LIN {X 0,Y 530.252,Z 278.433,A -85,B 0,C 180,E1 -4543.36,E2 -4543.36} C_VEL
LIN {X 0,Y 527.412,Z 278.789,A -85,B 0,C 180,E1 -4544.388,E2 -4544.388} C_VEL
LIN {X 0,Y 525.021,Z 279.084,A -85,B 0,C 180,E1 -4545.217,E2 -4545.217} C_VEL
LIN {X 0,Y 523.993,Z 279.212,A -85,B 0,C 180,E1 -4545.856,E2 -4545.856} C_VEL
LIN {X 0,Y 523.909,Z 279.223,A -85,B 0,C 180,E1 -4546.072,E2 -4546.072} C_VEL
LIN {X 0,Y 523.934,Z 279.22,A -85,B 0,C 180,E1 -4548.907,E2 -4548.907} C_VEL
LIN {X 0,Y 523.909,Z 279.226,A -85,B 0,C 180,E1 -4551.897,E2 -4551.897} C_VEL
LIN {X 0,Y 523.93,Z 279.219,A -85,B 0,C 180,E1 -4554.908,E2 -4554.908} C_VEL
LIN {X 0,Y 523.934,Z 279.224,A -85,B 0,C 180,E1 -4557.677,E2 -4557.677} C_VEL
LIN {X 0,Y 523.96,Z 279.215,A -85,B 0,C 180,E1 -4560.672,E2 -4560.672} C_VEL
LIN {X 0,Y 523.968,Z 279.22,A -85,B 0,C 180,E1 -4563.728,E2 -4563.728} C_VEL
LIN {X 0,Y 523.926,Z 279.22,A -85,B 0,C 180,E1 -4566.27,E2 -4566.27} C_VEL
LIN {X 0,Y 523.937,Z 279.221,A -85,B 0,C 180,E1 -4568.766,E2 -4568.766} C_VEL
LIN {X 0,Y 523.943,Z 279.222,A -85,B 0,C 180,E1 -4571.22,E2 -4571.22} C_VEL
LIN {X 0,Y 523.925,Z 279.22,A -85,B 0,C 180,E1 -4573.638,E2 -4573.638} C_VEL
LIN {X 0,Y 523.928,Z 279.219,A -85,B 0,C 180,E1 -4576.028,E2 -4576.028} C_VEL
LIN {X 0,Y 524,Z 279.215,A -85,B 0,C 180,E1 -4578.394,E2 -4578.394} C_VEL
LIN {X 0,Y 523.986,Z 279.211,A -85,B 0,C 180,E1 -4581.516,E2 -4581.516} C_VEL
LIN {X 0,Y 524.058,Z 279.206,A -85,B 0,C 180,E1 -4584.613,E2 -4584.613} C_VEL
LIN {X 0,Y 524.093,Z 279.2,A -85,B 0,C 180,E1 -4587.694,E2 -4587.694} C_VEL
LIN {X 0,Y 524.084,Z 279.207,A -85,B 0,C 180,E1 -4590,E2 -4590} C_VEL
LIN {X 0,Y 524.093,Z 279.2,A -85,B 0,C 180,E1 -4592.306,E2 -4592.306} C_VEL
LIN {X 0,Y 524.059,Z 279.206,A -85,B 0,C 180,E1 -4595.387,E2 -4595.387} C_VEL
LIN {X 0,Y 523.986,Z 279.211,A -85,B 0,C 180,E1 -4598.484,E2 -4598.484} C_VEL
LIN {X 0,Y 523.99,Z 279.214,A -85,B 0,C 180,E1 -4601.74,E2 -4601.74} C_VEL
LIN {X 0,Y 523.981,Z 279.218,A -85,B 0,C 180,E1 -4605.053,E2 -4605.053} C_VEL
LIN {X 0,Y 523.953,Z 279.216,A -85,B 0,C 180,E1 -4607.969,E2 -4607.969} C_VEL
LIN {X 0,Y 523.962,Z 279.218,A -85,B 0,C 180,E1 -4610.411,E2 -4610.411} C_VEL
LIN {X 0,Y 523.906,Z 279.227,A -85,B 0,C 180,E1 -4612.894,E2 -4612.894} C_VEL
LIN {X 0,Y 523.945,Z 279.217,A -85,B 0,C 180,E1 -4615.419,E2 -4615.419} C_VEL
LIN {X 0,Y 523.961,Z 279.219,A -85,B 0,C 180,E1 -4618,E2 -4618} C_VEL
LIN {X 0,Y 523.943,Z 279.219,A -85,B 0,C 180,E1 -4620.857,E2 -4620.857} C_VEL
LIN {X 0,Y 523.954,Z 279.22,A -85,B 0,C 180,E1 -4623.736,E2 -4623.736} C_VEL
LIN {X 0,Y 523.914,Z 279.223,A -85,B 0,C 180,E1 -4626.405,E2 -4626.405} C_VEL
LIN {X 0,Y 523.915,Z 279.222,A -85,B 0,C 180,E1 -4629.086,E2 -4629.086} C_VEL
LIN {X 0,Y 523.945,Z 279.219,A -85,B 0,C 180,E1 -4632.12,E2 -4632.12} C_VEL
LIN {X 0,Y 523.931,Z 279.226,A -85,B 0,C 180,E1 -4635.312,E2 -4635.312} C_VEL
LIN {X 0,Y 523.932,Z 279.22,A -85,B 0,C 180,E1 -4638.693,E2 -4638.693} C_VEL
LIN {X 0,Y 523.906,Z 279.221,A -85,B 0,C 180,E1 -4641.899,E2 -4641.899} C_VEL
LIN {X 0,Y 523.908,Z 279.227,A -85,B 0,C 180,E1 -4644.914,E2 -4644.914} C_VEL
LIN {X 0,Y 523.925,Z 279.218,A -85,B 0,C 180,E1 -4647.682,E2 -4647.682} C_VEL
LIN {X 0,Y 524.01,Z 279.336,A -85,B 0,C 180,E1 -4650.028,E2 -4650.028} C_VEL
LIN {X 0,Y 523.881,Z 285.472,A -85,B 0,C 180,E1 -4652.865,E2 -4652.865} C_VEL
LIN {X 0,Y 523.769,Z 291.976,A -85,B 0,C 180,E1 -4655.844,E2 -4655.844} C_VEL
LIN {X 0,Y 523.697,Z 298.443,A -85,B 0,C 180,E1 -4658.757,E2 -4658.757} C_VEL
LIN {X 0,Y 523.615,Z 303.894,A -85,B 0,C 180,E1 -4661.209,E2 -4661.209} C_VEL
LIN {X 0,Y 523.527,Z 309.386,A -85,B 0,C 180,E1 -4663.627,E2 -4663.627} C_VEL
LIN {X 0,Y 523.496,Z 314.819,A -85,B 0,C 180,E1 -4666.017,E2 -4666.017} C_VEL
LIN {X 0,Y 523.482,Z 320.596,A -85,B 0,C 180,E1 -4668.54,E2 -4668.54} C_VEL
LIN {X 0,Y 523.415,Z 328.516,A -85,B 0,C 180,E1 -4671.969,E2 -4671.969} C_VEL
LIN {X 0,Y 524.16,Z 336.561,A -85,B 0,C 180,E1 -4672.296,E2 -4672.296} C_VEL
LIN {X 0,Y 523.983,Z 346.121,A -85,B 0,C 180,E1 -4672.807,E2 -4672.807} C_VEL
LIN {X 0,Y 523.913,Z 353.385,A -85,B 0,C 180,E1 -4673.324,E2 -4673.324} C_VEL
LIN {X 0,Y 523.776,Z 359.239,A -85,B 0,C 180,E1 -4673.839,E2 -4673.839} C_VEL
LIN {X 0,Y 523.715,Z 366.141,A -85,B 0,C 180,E1 -4674.611,E2 -4674.611} C_VEL
LIN {X 0,Y 523.612,Z 371.545,A -85,B 0,C 180,E1 -4675.382,E2 -4675.382} C_VEL
LIN {X 0,Y 523.571,Z 375.823,A -85,B 0,C 180,E1 -4676.153,E2 -4676.153} C_VEL
LIN {X 0,Y 523.482,Z 379.147,A -85,B 0,C 180,E1 -4676.923,E2 -4676.923} C_VEL
LIN {X 0,Y 523.384,Z 381.639,A -85,B 0,C 180,E1 -4677.692,E2 -4677.692} C_VEL
LIN {X 0,Y 523.335,Z 383.365,A -85,B 0,C 180,E1 -4678.462,E2 -4678.462} C_VEL
LIN {X 0,Y 523.326,Z 384.379,A -85,B 0,C 180,E1 -4679.232,E2 -4679.232} C_VEL
LIN {X 0,Y 523.327,Z 384.776,A -85,B 0,C 180,E1 -4680.001,E2 -4680.001} C_VEL
LIN {X 0,Y 523.33,Z 384.536,A -85,B 0,C 180,E1 -4680.77,E2 -4680.77} C_VEL
LIN {X 0,Y 523.344,Z 383.632,A -85,B 0,C 180,E1 -4681.54,E2 -4681.54} C_VEL
LIN {X 0,Y 523.49,Z 380.907,A -85,B 0,C 180,E1 -4682.694,E2 -4682.694} C_VEL
LIN {X 0,Y 523.588,Z 378.19,A -85,B 0,C 180,E1 -4683.464,E2 -4683.464} C_VEL
LIN {X 0,Y 523.626,Z 373.539,A -85,B 0,C 180,E1 -4684.427,E2 -4684.427} C_VEL
LIN {X 0,Y 523.724,Z 368.666,A -85,B 0,C 180,E1 -4685.198,E2 -4685.198} C_VEL
LIN {X 0,Y 523.808,Z 362.441,A -85,B 0,C 180,E1 -4685.969,E2 -4685.969} C_VEL
LIN {X 0,Y 523.994,Z 354.754,A -85,B 0,C 180,E1 -4686.702,E2 -4686.702} C_VEL
LIN {X 0,Y 524.043,Z 346.949,A -85,B 0,C 180,E1 -4687.282,E2 -4687.282} C_VEL
LIN {X 0,Y 524.218,Z 337.48,A -85,B 0,C 180,E1 -4687.802,E2 -4687.802} C_VEL
LIN {X 0,Y 523.898,Z 331.555,A -85,B 0,C 180,E1 -4688.05,E2 -4688.05} C_VEL
LIN {X 0,Y 523.497,Z 329.053,A -85,B 0,C 180,E1 -4688.153,E2 -4688.153} C_VEL
LIN {X 0,Y 523.539,Z 321.18,A -85,B 0,C 180,E1 -4691.617,E2 -4691.617} C_VEL
LIN {X 0,Y 523.658,Z 313.899,A -85,B 0,C 180,E1 -4694.914,E2 -4694.914} C_VEL
LIN {X 0,Y 523.734,Z 307.092,A -85,B 0,C 180,E1 -4697.978,E2 -4697.978} C_VEL
LIN {X 0,Y 523.84,Z 301.836,A -85,B 0,C 180,E1 -4700.416,E2 -4700.416} C_VEL
LIN {X 0,Y 523.889,Z 296.392,A -85,B 0,C 180,E1 -4702.895,E2 -4702.895} C_VEL
LIN {X 0,Y 524.057,Z 289.588,A -85,B 0,C 180,E1 -4706.035,E2 -4706.035} C_VEL
LIN {X 0,Y 524.173,Z 283.477,A -85,B 0,C 180,E1 -4708.861,E2 -4708.861} C_VEL
LIN {X 0,Y 523.971,Z 279.222,A -85,B 0,C 180,E1 -4710.918,E2 -4710.918} C_VEL
LIN {X 0,Y 523.965,Z 279.222,A -85,B 0,C 180,E1 -4713.735,E2 -4713.735} C_VEL
LIN {X 0,Y 523.909,Z 279.227,A -85,B 0,C 180,E1 -4716.402,E2 -4716.402} C_VEL
LIN {X 0,Y 523.925,Z 279.227,A -85,B 0,C 180,E1 -4719.085,E2 -4719.085} C_VEL
LIN {X 0,Y 523.957,Z 279.222,A -85,B 0,C 180,E1 -4722.119,E2 -4722.119} C_VEL
LIN {X 0,Y 523.949,Z 279.223,A -85,B 0,C 180,E1 -4725.31,E2 -4725.31} C_VEL
LIN {X 0,Y 523.961,Z 279.222,A -85,B 0,C 180,E1 -4728.69,E2 -4728.69} C_VEL
LIN {X 0,Y 523.921,Z 279.226,A -85,B 0,C 180,E1 -4731.081,E2 -4731.081} C_VEL
LIN {X 0,Y 523.905,Z 279.229,A -85,B 0,C 180,E1 -4733.825,E2 -4733.825} C_VEL
LIN {X 0,Y 523.946,Z 279.225,A -85,B 0,C 180,E1 -4736.636,E2 -4736.636} C_VEL
LIN {X 0,Y 523.932,Z 279.256,A -85,B 0,C 180,E1 -4738.791,E2 -4738.791} C_VEL
LIN {X 0,Y 525.748,Z 287.197,A -85,B 0,C 180,E1 -4740.835,E2 -4740.835} C_VEL
LIN {X 0,Y 526.442,Z 291.224,A -85,B 0,C 180,E1 -4741.776,E2 -4741.776} C_VEL
LIN {X 0,Y 525.737,Z 304.415,A -85,B 0,C 180,E1 -4744.462,E2 -4744.462} C_VEL
LIN {X 0,Y 525.131,Z 318.686,A -85,B 0,C 180,E1 -4747.163,E2 -4747.163} C_VEL
LIN {X 0,Y 524.702,Z 334.54,A -85,B 0,C 180,E1 -4750.028,E2 -4750.028} C_VEL
LIN {X 0,Y 524.357,Z 350.704,A -85,B 0,C 180,E1 -4752.85,E2 -4752.85} C_VEL
LIN {X 0,Y 524.062,Z 369.627,A -85,B 0,C 180,E1 -4756.031,E2 -4756.031} C_VEL
LIN {X 0,Y 524.024,Z 371.591,A -85,B 0,C 180,E1 -4756.339,E2 -4756.339} C_VEL
LIN {X 0,Y 525.306,Z 382.111,A -85,B 0,C 180,E1 -4756.558,E2 -4756.558} C_VEL
LIN {X 0,Y 525.125,Z 394.093,A -85,B 0,C 180,E1 -4756.898,E2 -4756.898} C_VEL
LIN {X 0,Y 524.847,Z 407.07,A -85,B 0,C 180,E1 -4757.432,E2 -4757.432} C_VEL
LIN {X 0,Y 524.626,Z 419.038,A -85,B 0,C 180,E1 -4758.09,E2 -4758.09} C_VEL
LIN {X 0,Y 524.366,Z 430.416,A -85,B 0,C 180,E1 -4758.892,E2 -4758.892} C_VEL
LIN {X 0,Y 524.109,Z 440.369,A -85,B 0,C 180,E1 -4759.766,E2 -4759.766} C_VEL
LIN {X 0,Y 523.897,Z 449.423,A -85,B 0,C 180,E1 -4760.736,E2 -4760.736} C_VEL
LIN {X 0,Y 523.699,Z 458.25,A -85,B 0,C 180,E1 -4761.899,E2 -4761.899} C_VEL
LIN {X 0,Y 523.576,Z 465.285,A -85,B 0,C 180,E1 -4763.061,E2 -4763.061} C_VEL
LIN {X 0,Y 523.524,Z 470.919,A -85,B 0,C 180,E1 -4764.221,E2 -4764.221} C_VEL
LIN {X 0,Y 523.361,Z 475.325,A -85,B 0,C 180,E1 -4765.379,E2 -4765.379} C_VEL
LIN {X 0,Y 523.444,Z 477.673,A -85,B 0,C 180,E1 -4766.151,E2 -4766.151} C_VEL
LIN {X 0,Y 523.368,Z 479.561,A -85,B 0,C 180,E1 -4766.921,E2 -4766.921} C_VEL
LIN {X 0,Y 523.336,Z 480.978,A -85,B 0,C 180,E1 -4767.691,E2 -4767.691} C_VEL
LIN {X 0,Y 523.25,Z 482.598,A -85,B 0,C 180,E1 -4769.23,E2 -4769.23} C_VEL
LIN {X 0,Y 523.246,Z 482.818,A -85,B 0,C 180,E1 -4770,E2 -4770} C_VEL
LIN {X 0,Y 523.25,Z 482.599,A -85,B 0,C 180,E1 -4770.77,E2 -4770.77} C_VEL
LIN {X 0,Y 523.336,Z 480.979,A -85,B 0,C 180,E1 -4772.309,E2 -4772.309} C_VEL
LIN {X 0,Y 523.368,Z 479.563,A -85,B 0,C 180,E1 -4773.079,E2 -4773.079} C_VEL
LIN {X 0,Y 523.425,Z 476.591,A -85,B 0,C 180,E1 -4774.235,E2 -4774.235} C_VEL
LIN {X 0,Y 523.464,Z 472.56,A -85,B 0,C 180,E1 -4775.393,E2 -4775.393} C_VEL
LIN {X 0,Y 523.524,Z 467.22,A -85,B 0,C 180,E1 -4776.58,E2 -4776.58} C_VEL
LIN {X 0,Y 523.666,Z 460.813,A -85,B 0,C 180,E1 -4777.713,E2 -4777.713} C_VEL
LIN {X 0,Y 523.846,Z 452.653,A -85,B 0,C 180,E1 -4778.875,E2 -4778.875} C_VEL
LIN {X 0,Y 524.015,Z 444.319,A -85,B 0,C 180,E1 -4779.846,E2 -4779.846} C_VEL
LIN {X 0,Y 524.305,Z 434.143,A -85,B 0,C 180,E1 -4780.816,E2 -4780.816} C_VEL
LIN {X 0,Y 524.583,Z 422.543,A -85,B 0,C 180,E1 -4781.694,E2 -4781.694} C_VEL
LIN {X 0,Y 524.803,Z 411.237,A -85,B 0,C 180,E1 -4782.373,E2 -4782.373} C_VEL
LIN {X 0,Y 524.996,Z 399.713,A -85,B 0,C 180,E1 -4782.908,E2 -4782.908} C_VEL
LIN {X 0,Y 525.219,Z 386.487,A -85,B 0,C 180,E1 -4783.346,E2 -4783.346} C_VEL
LIN {X 0,Y 525.058,Z 379.612,A -85,B 0,C 180,E1 -4783.513,E2 -4783.513} C_VEL
LIN {X 0,Y 524.023,Z 371.416,A -85,B 0,C 180,E1 -4783.698,E2 -4783.698} C_VEL
LIN {X 0,Y 524.364,Z 353.595,A -85,B 0,C 180,E1 -4786.748,E2 -4786.748} C_VEL
LIN {X 0,Y 524.721,Z 336.251,A -85,B 0,C 180,E1 -4789.767,E2 -4789.767} C_VEL
LIN {X 0,Y 525.162,Z 320.599,A -85,B 0,C 180,E1 -4792.571,E2 -4792.571} C_VEL
LIN {X 0,Y 525.672,Z 305.612,A -85,B 0,C 180,E1 -4795.33,E2 -4795.33} C_VEL
LIN {X 0,Y 526.257,Z 292.199,A -85,B 0,C 180,E1 -4797.867,E2 -4797.867} C_VEL
LIN {X 0,Y 526.162,Z 289.475,A -85,B 0,C 180,E1 -4798.403,E2 -4798.403} C_VEL
LIN {X 0,Y 523.946,Z 279.223,A -85,B 0,C 180,E1 -4800.589,E2 -4800.589} C_VEL
LIN {X 0,Y 523.934,Z 279.224,A -85,B 0,C 180,E1 -4803.729,E2 -4803.729} C_VEL
LIN {X 0,Y 523.908,Z 279.229,A -85,B 0,C 180,E1 -4806.401,E2 -4806.401} C_VEL
LIN {X 0,Y 523.926,Z 279.224,A -85,B 0,C 180,E1 -4809.084,E2 -4809.084} C_VEL
LIN {X 0,Y 523.956,Z 279.221,A -85,B 0,C 180,E1 -4812.119,E2 -4812.119} C_VEL
LIN {X 0,Y 523.96,Z 279.22,A -85,B 0,C 180,E1 -4815.309,E2 -4815.309} C_VEL
LIN {X 0,Y 523.961,Z 279.22,A -85,B 0,C 180,E1 -4818.69,E2 -4818.69} C_VEL
LIN {X 0,Y 523.924,Z 279.226,A -85,B 0,C 180,E1 -4821.08,E2 -4821.08} C_VEL
LIN {X 0,Y 523.906,Z 279.227,A -85,B 0,C 180,E1 -4823.825,E2 -4823.825} C_VEL
LIN {X 0,Y 523.919,Z 279.229,A -85,B 0,C 180,E1 -4826.633,E2 -4826.633} C_VEL
LIN {X 0,Y 523.954,Z 279.223,A -85,B 0,C 180,E1 -4829.355,E2 -4829.355} C_VEL
LIN {X 0,Y 523.678,Z 279.26,A -85,B 0,C 180,E1 -4831.765,E2 -4831.765} C_VEL
LIN {X 0,Y 523.641,Z 279.581,A -85,B 0,C 180,E1 -4831.981,E2 -4831.981} C_VEL
LIN {X 0,Y 523.628,Z 288.099,A -85,B 0,C 180,E1 -4834.989,E2 -4834.989} C_VEL
LIN {X 0,Y 523.644,Z 295.888,A -85,B 0,C 180,E1 -4837.926,E2 -4837.926} C_VEL
LIN {X 0,Y 523.627,Z 303.05,A -85,B 0,C 180,E1 -4840.801,E2 -4840.801} C_VEL
LIN {X 0,Y 523.607,Z 310.075,A -85,B 0,C 180,E1 -4843.627,E2 -4843.627} C_VEL
LIN {X 0,Y 523.578,Z 315.757,A -85,B 0,C 180,E1 -4846.017,E2 -4846.017} C_VEL
LIN {X 0,Y 523.578,Z 323.144,A -85,B 0,C 180,E1 -4849.168,E2 -4849.168} C_VEL
LIN {X 0,Y 523.519,Z 329.885,A -85,B 0,C 180,E1 -4852.066,E2 -4852.066} C_VEL
LIN {X 0,Y 524.115,Z 337.803,A -85,B 0,C 180,E1 -4852.39,E2 -4852.39} C_VEL
LIN {X 0,Y 523.977,Z 346.945,A -85,B 0,C 180,E1 -4852.872,E2 -4852.872} C_VEL
LIN {X 0,Y 523.889,Z 354.734,A -85,B 0,C 180,E1 -4853.44,E2 -4853.44} C_VEL
LIN {X 0,Y 523.709,Z 361.132,A -85,B 0,C 180,E1 -4854.029,E2 -4854.029} C_VEL
LIN {X 0,Y 523.725,Z 367.73,A -85,B 0,C 180,E1 -4854.802,E2 -4854.802} C_VEL
LIN {X 0,Y 523.607,Z 373.909,A -85,B 0,C 180,E1 -4855.765,E2 -4855.765} C_VEL
LIN {X 0,Y 523.585,Z 377.692,A -85,B 0,C 180,E1 -4856.536,E2 -4856.536} C_VEL
LIN {X 0,Y 523.489,Z 380.55,A -85,B 0,C 180,E1 -4857.306,E2 -4857.306} C_VEL
LIN {X 0,Y 523.338,Z 383.385,A -85,B 0,C 180,E1 -4858.46,E2 -4858.46} C_VEL
LIN {X 0,Y 523.324,Z 384.42,A -85,B 0,C 180,E1 -4859.23,E2 -4859.23} C_VEL
LIN {X 0,Y 523.321,Z 384.784,A -85,B 0,C 180,E1 -4859.999,E2 -4859.999} C_VEL
LIN {X 0,Y 523.322,Z 384.485,A -85,B 0,C 180,E1 -4860.768,E2 -4860.768} C_VEL
LIN {X 0,Y 523.333,Z 383.517,A -85,B 0,C 180,E1 -4861.538,E2 -4861.538} C_VEL
LIN {X 0,Y 523.489,Z 380.73,A -85,B 0,C 180,E1 -4862.692,E2 -4862.692} C_VEL
LIN {X 0,Y 523.521,Z 377.963,A -85,B 0,C 180,E1 -4863.462,E2 -4863.462} C_VEL
LIN {X 0,Y 523.624,Z 373.194,A -85,B 0,C 180,E1 -4864.425,E2 -4864.425} C_VEL
LIN {X 0,Y 523.668,Z 368.214,A -85,B 0,C 180,E1 -4865.196,E2 -4865.196} C_VEL
LIN {X 0,Y 523.692,Z 361.85,A -85,B 0,C 180,E1 -4865.969,E2 -4865.969} C_VEL
LIN {X 0,Y 523.899,Z 354.1,A -85,B 0,C 180,E1 -4866.685,E2 -4866.685} C_VEL
LIN {X 0,Y 523.983,Z 344.972,A -85,B 0,C 180,E1 -4867.319,E2 -4867.319} C_VEL
LIN {X 0,Y 524.107,Z 336.379,A -85,B 0,C 180,E1 -4867.754,E2 -4867.754} C_VEL
LIN {X 0,Y 523.469,Z 329.487,A -85,B 0,C 180,E1 -4868.03,E2 -4868.03} C_VEL
LIN {X 0,Y 523.536,Z 322.935,A -85,B 0,C 180,E1 -4870.831,E2 -4870.831} C_VEL
LIN {X 0,Y 523.557,Z 315.551,A -85,B 0,C 180,E1 -4873.981,E2 -4873.981} C_VEL
LIN {X 0,Y 523.585,Z 309.972,A -85,B 0,C 180,E1 -4876.371,E2 -4876.371} C_VEL
LIN {X 0,Y 523.63,Z 304.228,A -85,B 0,C 180,E1 -4878.79,E2 -4878.79} C_VEL
LIN {X 0,Y 523.683,Z 298.544,A -85,B 0,C 180,E1 -4881.243,E2 -4881.243} C_VEL
LIN {X 0,Y 523.722,Z 291.706,A -85,B 0,C 180,E1 -4884.144,E2 -4884.144} C_VEL
LIN {X 0,Y 523.739,Z 284.504,A -85,B 0,C 180,E1 -4887.143,E2 -4887.143} C_VEL
LIN {X 0,Y 523.863,Z 279.235,A -85,B 0,C 180,E1 -4889.361,E2 -4889.361} C_VEL
LIN {X 0,Y 523.924,Z 279.218,A -85,B 0,C 180,E1 -4892.449,E2 -4892.449} C_VEL
LIN {X 0,Y 523.907,Z 279.228,A -85,B 0,C 180,E1 -4895.226,E2 -4895.226} C_VEL
LIN {X 0,Y 523.906,Z 279.221,A -85,B 0,C 180,E1 -4898.101,E2 -4898.101} C_VEL
LIN {X 0,Y 523.932,Z 279.22,A -85,B 0,C 180,E1 -4901.307,E2 -4901.307} C_VEL
LIN {X 0,Y 523.931,Z 279.226,A -85,B 0,C 180,E1 -4904.688,E2 -4904.688} C_VEL
LIN {X 0,Y 523.909,Z 279.223,A -85,B 0,C 180,E1 -4906.072,E2 -4906.072} C_VEL
LIN {X 0,Y 523.239,Z 279.311,A -85,B 0,C 180,E1 -4906.715,E2 -4906.715} C_VEL
LIN {X 0,Y 520.385,Z 279.664,A -85,B 0,C 180,E1 -4907.758,E2 -4907.758} C_VEL
LIN {X 0,Y 517.979,Z 279.965,A -85,B 0,C 180,E1 -4908.597,E2 -4908.597} C_VEL
LIN {X 0,Y 516.954,Z 280.088,A -85,B 0,C 180,E1 -4909.246,E2 -4909.246} C_VEL
LIN {X 0,Y 516.874,Z 280.098,A -85,B 0,C 180,E1 -4909.466,E2 -4909.466} C_VEL
LIN {X 0,Y 516.857,Z 280.106,A -85,B 0,C 180,E1 -4912.273,E2 -4912.273} C_VEL
LIN {X 0,Y 516.887,Z 280.097,A -85,B 0,C 180,E1 -4915.175,E2 -4915.175} C_VEL
LIN {X 0,Y 516.874,Z 280.104,A -85,B 0,C 180,E1 -4917.975,E2 -4917.975} C_VEL
LIN {X 0,Y 516.926,Z 280.092,A -85,B 0,C 180,E1 -4920.696,E2 -4920.696} C_VEL
LIN {X 0,Y 516.935,Z 280.095,A -85,B 0,C 180,E1 -4923.802,E2 -4923.802} C_VEL
LIN {X 0,Y 516.862,Z 280.102,A -85,B 0,C 180,E1 -4926.776,E2 -4926.776} C_VEL
LIN {X 0,Y 516.928,Z 280.093,A -85,B 0,C 180,E1 -4929.731,E2 -4929.731} C_VEL
LIN {X 0,Y 516.917,Z 280.096,A -85,B 0,C 180,E1 -4932.596,E2 -4932.596} C_VEL
LIN {X 0,Y 516.93,Z 280.095,A -85,B 0,C 180,E1 -4935.03,E2 -4935.03} C_VEL
LIN {X 0,Y 516.953,Z 280.091,A -85,B 0,C 180,E1 -4938.233,E2 -4938.233} C_VEL
LIN {X 0,Y 516.95,Z 280.088,A -85,B 0,C 180,E1 -4941.399,E2 -4941.399} C_VEL
LIN {X 0,Y 517.005,Z 280.085,A -85,B 0,C 180,E1 -4944.54,E2 -4944.54} C_VEL
LIN {X 0,Y 517.062,Z 280.076,A -85,B 0,C 180,E1 -4947.663,E2 -4947.663} C_VEL
LIN {X 0,Y 517.052,Z 280.083,A -85,B 0,C 180,E1 -4950,E2 -4950} C_VEL
LIN {X 0,Y 517.063,Z 280.076,A -85,B 0,C 180,E1 -4952.337,E2 -4952.337} C_VEL
LIN {X 0,Y 517.006,Z 280.085,A -85,B 0,C 180,E1 -4955.46,E2 -4955.46} C_VEL
LIN {X 0,Y 516.951,Z 280.088,A -85,B 0,C 180,E1 -4958.601,E2 -4958.601} C_VEL
LIN {X 0,Y 516.939,Z 280.092,A -85,B 0,C 180,E1 -4961.807,E2 -4961.807} C_VEL
LIN {X 0,Y 516.932,Z 280.097,A -85,B 0,C 180,E1 -4965.147,E2 -4965.147} C_VEL
LIN {X 0,Y 516.915,Z 280.094,A -85,B 0,C 180,E1 -4968.223,E2 -4968.223} C_VEL
LIN {X 0,Y 516.902,Z 280.099,A -85,B 0,C 180,E1 -4970.702,E2 -4970.702} C_VEL
LIN {X 0,Y 516.901,Z 280.097,A -85,B 0,C 180,E1 -4974.073,E2 -4974.073} C_VEL
LIN {X 0,Y 516.919,Z 280.098,A -85,B 0,C 180,E1 -4976.658,E2 -4976.658} C_VEL
LIN {X 0,Y 516.915,Z 280.094,A -85,B 0,C 180,E1 -4979.527,E2 -4979.527} C_VEL
LIN {X 0,Y 516.892,Z 280.099,A -85,B 0,C 180,E1 -4982.545,E2 -4982.545} C_VEL
LIN {X 0,Y 516.875,Z 280.099,A -85,B 0,C 180,E1 -4985.333,E2 -4985.333} C_VEL
LIN {X 0,Y 516.873,Z 280.103,A -85,B 0,C 180,E1 -4987.944,E2 -4987.944} C_VEL
LIN {X 0,Y 516.876,Z 280.098,A -85,B 0,C 180,E1 -4990.743,E2 -4990.743} C_VEL
LIN {X 0,Y 516.874,Z 280.099,A -85,B 0,C 180,E1 -4992.833,E2 -4992.833} C_VEL
LIN {X 0,Y 516.887,Z 280.099,A -85,B 0,C 180,E1 -4995.008,E2 -4995.008} C_VEL
LIN {X 0,Y 516.895,Z 280.095,A -85,B 0,C 180,E1 -4998.401,E2 -4998.401} C_VEL
LIN {X 0,Y 516.869,Z 280.102,A -85,B 0,C 180,E1 -5001.285,E2 -5001.285} C_VEL
LIN {X 0,Y 516.85,Z 280.101,A -85,B 0,C 180,E1 -5004.22,E2 -5004.22} C_VEL
LIN {X 0,Y 516.874,Z 280.1,A -85,B 0,C 180,E1 -5007.053,E2 -5007.053} C_VEL
LIN {X 0,Y 516.986,Z 280.252,A -85,B 0,C 180,E1 -5010.009,E2 -5010.009} C_VEL
LIN {X 0,Y 516.88,Z 285.513,A -85,B 0,C 180,E1 -5012.466,E2 -5012.466} C_VEL
LIN {X 0,Y 516.738,Z 291.14,A -85,B 0,C 180,E1 -5015.064,E2 -5015.064} C_VEL
LIN {X 0,Y 516.683,Z 296.83,A -85,B 0,C 180,E1 -5017.661,E2 -5017.661} C_VEL
LIN {X 0,Y 516.598,Z 302.219,A -85,B 0,C 180,E1 -5020.118,E2 -5020.118} C_VEL
LIN {X 0,Y 516.523,Z 307.758,A -85,B 0,C 180,E1 -5022.583,E2 -5022.583} C_VEL
LIN {X 0,Y 516.439,Z 315.029,A -85,B 0,C 180,E1 -5025.822,E2 -5025.822} C_VEL
LIN {X 0,Y 516.426,Z 321.081,A -85,B 0,C 180,E1 -5028.478,E2 -5028.478} C_VEL
LIN {X 0,Y 516.368,Z 328.8,A -85,B 0,C 180,E1 -5031.834,E2 -5031.834} C_VEL
LIN {X 0,Y 517.171,Z 337.358,A -85,B 0,C 180,E1 -5032.191,E2 -5032.191} C_VEL
LIN {X 0,Y 516.978,Z 346.809,A -85,B 0,C 180,E1 -5032.709,E2 -5032.709} C_VEL
LIN {X 0,Y 516.892,Z 354.568,A -85,B 0,C 180,E1 -5033.279,E2 -5033.279} C_VEL
LIN {X 0,Y 516.675,Z 361.71,A -85,B 0,C 180,E1 -5033.95,E2 -5033.95} C_VEL
LIN {X 0,Y 516.655,Z 368.211,A -85,B 0,C 180,E1 -5034.733,E2 -5034.733} C_VEL
LIN {X 0,Y 516.585,Z 373.299,A -85,B 0,C 180,E1 -5035.514,E2 -5035.514} C_VEL
LIN {X 0,Y 516.53,Z 376.442,A -85,B 0,C 180,E1 -5036.1,E2 -5036.1} C_VEL
LIN {X 0,Y 516.422,Z 379.776,A -85,B 0,C 180,E1 -5036.881,E2 -5036.881} C_VEL
LIN {X 0,Y 516.32,Z 382.277,A -85,B 0,C 180,E1 -5037.661,E2 -5037.661} C_VEL
LIN {X 0,Y 516.269,Z 384.02,A -85,B 0,C 180,E1 -5038.441,E2 -5038.441} C_VEL
LIN {X 0,Y 516.259,Z 385.054,A -85,B 0,C 180,E1 -5039.221,E2 -5039.221} C_VEL
LIN {X 0,Y 516.261,Z 385.459,A -85,B 0,C 180,E1 -5040.001,E2 -5040.001} C_VEL
LIN {X 0,Y 516.265,Z 385.221,A -85,B 0,C 180,E1 -5040.781,E2 -5040.781} C_VEL
LIN {X 0,Y 516.28,Z 384.317,A -85,B 0,C 180,E1 -5041.561,E2 -5041.561} C_VEL
LIN {X 0,Y 516.444,Z 381.604,A -85,B 0,C 180,E1 -5042.731,E2 -5042.731} C_VEL
LIN {X 0,Y 516.557,Z 378.885,A -85,B 0,C 180,E1 -5043.511,E2 -5043.511} C_VEL
LIN {X 0,Y 516.592,Z 374.252,A -85,B 0,C 180,E1 -5044.488,E2 -5044.488} C_VEL
LIN {X 0,Y 516.702,Z 369.399,A -85,B 0,C 180,E1 -5045.269,E2 -5045.269} C_VEL
LIN {X 0,Y 516.798,Z 363.2,A -85,B 0,C 180,E1 -5046.051,E2 -5046.051} C_VEL
LIN {X 0,Y 517,Z 355.737,A -85,B 0,C 180,E1 -5046.78,E2 -5046.78} C_VEL
LIN {X 0,Y 517.065,Z 347.867,A -85,B 0,C 180,E1 -5047.381,E2 -5047.381} C_VEL
LIN {X 0,Y 517.252,Z 338.579,A -85,B 0,C 180,E1 -5047.908,E2 -5047.908} C_VEL
LIN {X 0,Y 516.761,Z 331.575,A -85,B 0,C 180,E1 -5048.211,E2 -5048.211} C_VEL
LIN {X 0,Y 516.436,Z 329.468,A -85,B 0,C 180,E1 -5048.315,E2 -5048.315} C_VEL
LIN {X 0,Y 516.501,Z 321.71,A -85,B 0,C 180,E1 -5051.778,E2 -5051.778} C_VEL
LIN {X 0,Y 516.621,Z 314.561,A -85,B 0,C 180,E1 -5055.012,E2 -5055.012} C_VEL
LIN {X 0,Y 516.718,Z 307.554,A -85,B 0,C 180,E1 -5058.231,E2 -5058.231} C_VEL
LIN {X 0,Y 516.816,Z 302.172,A -85,B 0,C 180,E1 -5060.706,E2 -5060.706} C_VEL
LIN {X 0,Y 516.891,Z 296.77,A -85,B 0,C 180,E1 -5063.223,E2 -5063.223} C_VEL
LIN {X 0,Y 517.067,Z 290.353,A -85,B 0,C 180,E1 -5066.223,E2 -5066.223} C_VEL
LIN {X 0,Y 517.207,Z 283.85,A -85,B 0,C 180,E1 -5069.288,E2 -5069.288} C_VEL
LIN {X 0,Y 516.915,Z 280.101,A -85,B 0,C 180,E1 -5071.165,E2 -5071.165} C_VEL
LIN {X 0,Y 516.914,Z 280.1,A -85,B 0,C 180,E1 -5073.966,E2 -5073.966} C_VEL
LIN {X 0,Y 516.882,Z 280.103,A -85,B 0,C 180,E1 -5076.746,E2 -5076.746} C_VEL
LIN {X 0,Y 516.887,Z 280.102,A -85,B 0,C 180,E1 -5079.722,E2 -5079.722} C_VEL
LIN {X 0,Y 516.917,Z 280.098,A -85,B 0,C 180,E1 -5081.776,E2 -5081.776} C_VEL
LIN {X 0,Y 516.9,Z 280.1,A -85,B 0,C 180,E1 -5085.007,E2 -5085.007} C_VEL
LIN {X 0,Y 516.918,Z 280.099,A -85,B 0,C 180,E1 -5088.399,E2 -5088.399} C_VEL
LIN {X 0,Y 516.885,Z 280.102,A -85,B 0,C 180,E1 -5091.284,E2 -5091.284} C_VEL
LIN {X 0,Y 516.876,Z 280.104,A -85,B 0,C 180,E1 -5094.22,E2 -5094.22} C_VEL
LIN {X 0,Y 516.9,Z 280.103,A -85,B 0,C 180,E1 -5097.053,E2 -5097.053} C_VEL
LIN {X 0,Y 516.912,Z 280.19,A -85,B 0,C 180,E1 -5098.379,E2 -5098.379} C_VEL
LIN {X 0,Y 518.982,Z 289.358,A -85,B 0,C 180,E1 -5100.823,E2 -5100.823} C_VEL
LIN {X 0,Y 519.63,Z 293.239,A -85,B 0,C 180,E1 -5101.746,E2 -5101.746} C_VEL
LIN {X 0,Y 518.846,Z 305.52,A -85,B 0,C 180,E1 -5104.313,E2 -5104.313} C_VEL
LIN {X 0,Y 518.147,Z 319.92,A -85,B 0,C 180,E1 -5107.113,E2 -5107.113} C_VEL
LIN {X 0,Y 517.723,Z 334.692,A -85,B 0,C 180,E1 -5109.821,E2 -5109.821} C_VEL
LIN {X 0,Y 517.294,Z 351.397,A -85,B 0,C 180,E1 -5112.813,E2 -5112.813} C_VEL
LIN {X 0,Y 516.989,Z 369.028,A -85,B 0,C 180,E1 -5115.836,E2 -5115.836} C_VEL
LIN {X 0,Y 516.971,Z 371.058,A -85,B 0,C 180,E1 -5116.187,E2 -5116.187} C_VEL
LIN {X 0,Y 518.262,Z 383.091,A -85,B 0,C 180,E1 -5116.447,E2 -5116.447} C_VEL
LIN {X 0,Y 518.064,Z 396.509,A -85,B 0,C 180,E1 -5116.866,E2 -5116.866} C_VEL
LIN {X 0,Y 517.805,Z 407.77,A -85,B 0,C 180,E1 -5117.358,E2 -5117.358} C_VEL
LIN {X 0,Y 517.58,Z 419.197,A -85,B 0,C 180,E1 -5118.007,E2 -5118.007} C_VEL
LIN {X 0,Y 517.289,Z 430.61,A -85,B 0,C 180,E1 -5118.837,E2 -5118.837} C_VEL
LIN {X 0,Y 517.011,Z 441.435,A -85,B 0,C 180,E1 -5119.821,E2 -5119.821} C_VEL
LIN {X 0,Y 516.791,Z 450.212,A -85,B 0,C 180,E1 -5120.805,E2 -5120.805} C_VEL
LIN {X 0,Y 516.606,Z 458.713,A -85,B 0,C 180,E1 -5121.984,E2 -5121.984} C_VEL
LIN {X 0,Y 516.508,Z 464.527,A -85,B 0,C 180,E1 -5122.966,E2 -5122.966} C_VEL
LIN {X 0,Y 516.435,Z 470.189,A -85,B 0,C 180,E1 -5124.142,E2 -5124.142} C_VEL
LIN {X 0,Y 516.279,Z 474.62,A -85,B 0,C 180,E1 -5125.315,E2 -5125.315} C_VEL
LIN {X 0,Y 516.37,Z 476.979,A -85,B 0,C 180,E1 -5126.098,E2 -5126.098} C_VEL
LIN {X 0,Y 516.313,Z 478.884,A -85,B 0,C 180,E1 -5126.879,E2 -5126.879} C_VEL
LIN {X 0,Y 516.262,Z 480.308,A -85,B 0,C 180,E1 -5127.659,E2 -5127.659} C_VEL
LIN {X 0,Y 516.18,Z 481.94,A -85,B 0,C 180,E1 -5129.22,E2 -5129.22} C_VEL
LIN {X 0,Y 516.177,Z 482.165,A -85,B 0,C 180,E1 -5130,E2 -5130} C_VEL
LIN {X 0,Y 516.179,Z 481.947,A -85,B 0,C 180,E1 -5130.78,E2 -5130.78} C_VEL
LIN {X 0,Y 516.262,Z 480.326,A -85,B 0,C 180,E1 -5132.341,E2 -5132.341} C_VEL
LIN {X 0,Y 516.313,Z 478.91,A -85,B 0,C 180,E1 -5133.121,E2 -5133.121} C_VEL
LIN {X 0,Y 516.348,Z 475.93,A -85,B 0,C 180,E1 -5134.293,E2 -5134.293} C_VEL
LIN {X 0,Y 516.403,Z 471.888,A -85,B 0,C 180,E1 -5135.467,E2 -5135.467} C_VEL
LIN {X 0,Y 516.484,Z 465.83,A -85,B 0,C 180,E1 -5136.803,E2 -5136.803} C_VEL
LIN {X 0,Y 516.606,Z 458.837,A -85,B 0,C 180,E1 -5138.016,E2 -5138.016} C_VEL
LIN {X 0,Y 516.791,Z 450.378,A -85,B 0,C 180,E1 -5139.195,E2 -5139.195} C_VEL
LIN {X 0,Y 517.012,Z 441.647,A -85,B 0,C 180,E1 -5140.179,E2 -5140.179} C_VEL
LIN {X 0,Y 517.308,Z 430.883,A -85,B 0,C 180,E1 -5141.163,E2 -5141.163} C_VEL
LIN {X 0,Y 517.598,Z 419.58,A -85,B 0,C 180,E1 -5141.991,E2 -5141.991} C_VEL
LIN {X 0,Y 517.845,Z 408.227,A -85,B 0,C 180,E1 -5142.641,E2 -5142.641} C_VEL
LIN {X 0,Y 518.104,Z 395.767,A -85,B 0,C 180,E1 -5143.183,E2 -5143.183} C_VEL
LIN {X 0,Y 518.319,Z 382.944,A -85,B 0,C 180,E1 -5143.577,E2 -5143.577} C_VEL
LIN {X 0,Y 516.968,Z 371.19,A -85,B 0,C 180,E1 -5143.838,E2 -5143.838} C_VEL
LIN {X 0,Y 517.323,Z 354.315,A -85,B 0,C 180,E1 -5146.78,E2 -5146.78} C_VEL
LIN {X 0,Y 517.788,Z 335.183,A -85,B 0,C 180,E1 -5150.191,E2 -5150.191} C_VEL
LIN {X 0,Y 518.394,Z 316.746,A -85,B 0,C 180,E1 -5153.574,E2 -5153.574} C_VEL
LIN {X 0,Y 519.029,Z 301.065,A -85,B 0,C 180,E1 -5156.541,E2 -5156.541} C_VEL
LIN {X 0,Y 519.324,Z 291.538,A -85,B 0,C 180,E1 -5158.4,E2 -5158.4} C_VEL
LIN {X 0,Y 516.901,Z 280.101,A -85,B 0,C 180,E1 -5160.893,E2 -5160.893} C_VEL
LIN {X 0,Y 516.89,Z 280.102,A -85,B 0,C 180,E1 -5163.962,E2 -5163.962} C_VEL
LIN {X 0,Y 516.881,Z 280.102,A -85,B 0,C 180,E1 -5166.746,E2 -5166.746} C_VEL
LIN {X 0,Y 516.887,Z 280.102,A -85,B 0,C 180,E1 -5169.721,E2 -5169.721} C_VEL
LIN {X 0,Y 516.917,Z 280.099,A -85,B 0,C 180,E1 -5171.775,E2 -5171.775} C_VEL
LIN {X 0,Y 516.929,Z 280.097,A -85,B 0,C 180,E1 -5175.01,E2 -5175.01} C_VEL
LIN {X 0,Y 516.919,Z 280.097,A -85,B 0,C 180,E1 -5178.399,E2 -5178.399} C_VEL
LIN {X 0,Y 516.887,Z 280.102,A -85,B 0,C 180,E1 -5181.284,E2 -5181.284} C_VEL
LIN {X 0,Y 516.876,Z 280.103,A -85,B 0,C 180,E1 -5184.219,E2 -5184.219} C_VEL
LIN {X 0,Y 516.887,Z 280.103,A -85,B 0,C 180,E1 -5187.052,E2 -5187.052} C_VEL
LIN {X 0,Y 516.862,Z 280.107,A -85,B 0,C 180,E1 -5189.794,E2 -5189.794} C_VEL
LIN {X 0,Y 516.608,Z 280.195,A -85,B 0,C 180,E1 -5191.907,E2 -5191.907} C_VEL
LIN {X 0,Y 516.569,Z 287.931,A -85,B 0,C 180,E1 -5194.623,E2 -5194.623} C_VEL
LIN {X 0,Y 516.616,Z 295.888,A -85,B 0,C 180,E1 -5197.609,E2 -5197.609} C_VEL
LIN {X 0,Y 516.613,Z 303.307,A -85,B 0,C 180,E1 -5200.53,E2 -5200.53} C_VEL
LIN {X 0,Y 516.539,Z 310.17,A -85,B 0,C 180,E1 -5203.397,E2 -5203.397} C_VEL
LIN {X 0,Y 516.554,Z 316.156,A -85,B 0,C 180,E1 -5205.823,E2 -5205.823} C_VEL
LIN {X 0,Y 516.541,Z 323.683,A -85,B 0,C 180,E1 -5209.018,E2 -5209.018} C_VEL
LIN {X 0,Y 516.51,Z 330.79,A -85,B 0,C 180,E1 -5211.982,E2 -5211.982} C_VEL
LIN {X 0,Y 517.1,Z 337.286,A -85,B 0,C 180,E1 -5212.237,E2 -5212.237} C_VEL
LIN {X 0,Y 516.967,Z 345.857,A -85,B 0,C 180,E1 -5212.677,E2 -5212.677} C_VEL
LIN {X 0,Y 516.888,Z 354.442,A -85,B 0,C 180,E1 -5213.274,E2 -5213.274} C_VEL
LIN {X 0,Y 516.675,Z 361.749,A -85,B 0,C 180,E1 -5213.948,E2 -5213.948} C_VEL
LIN {X 0,Y 516.7,Z 368.366,A -85,B 0,C 180,E1 -5214.731,E2 -5214.731} C_VEL
LIN {X 0,Y 516.59,Z 373.439,A -85,B 0,C 180,E1 -5215.512,E2 -5215.512} C_VEL
LIN {X 0,Y 516.554,Z 378.345,A -85,B 0,C 180,E1 -5216.489,E2 -5216.489} C_VEL
LIN {X 0,Y 516.443,Z 381.21,A -85,B 0,C 180,E1 -5217.269,E2 -5217.269} C_VEL
LIN {X 0,Y 516.272,Z 384.047,A -85,B 0,C 180,E1 -5218.439,E2 -5218.439} C_VEL
LIN {X 0,Y 516.257,Z 385.081,A -85,B 0,C 180,E1 -5219.219,E2 -5219.219} C_VEL
LIN {X 0,Y 516.252,Z 385.442,A -85,B 0,C 180,E1 -5219.999,E2 -5219.999} C_VEL
LIN {X 0,Y 516.253,Z 385.137,A -85,B 0,C 180,E1 -5220.779,E2 -5220.779} C_VEL
LIN {X 0,Y 516.266,Z 384.161,A -85,B 0,C 180,E1 -5221.559,E2 -5221.559} C_VEL
LIN {X 0,Y 516.442,Z 381.355,A -85,B 0,C 180,E1 -5222.729,E2 -5222.729} C_VEL
LIN {X 0,Y 516.464,Z 378.577,A -85,B 0,C 180,E1 -5223.51,E2 -5223.51} C_VEL
LIN {X 0,Y 516.586,Z 373.789,A -85,B 0,C 180,E1 -5224.486,E2 -5224.486} C_VEL
LIN {X 0,Y 516.63,Z 368.786,A -85,B 0,C 180,E1 -5225.267,E2 -5225.267} C_VEL
LIN {X 0,Y 516.655,Z 362.395,A -85,B 0,C 180,E1 -5226.05,E2 -5226.05} C_VEL
LIN {X 0,Y 516.858,Z 355.502,A -85,B 0,C 180,E1 -5226.702,E2 -5226.702} C_VEL
LIN {X 0,Y 516.958,Z 347.129,A -85,B 0,C 180,E1 -5227.321,E2 -5227.321} C_VEL
LIN {X 0,Y 517.02,Z 337.893,A -85,B 0,C 180,E1 -5227.811,E2 -5227.811} C_VEL
LIN {X 0,Y 516.841,Z 333.024,A -85,B 0,C 180,E1 -5228.011,E2 -5228.011} C_VEL
LIN {X 0,Y 516.44,Z 330.044,A -85,B 0,C 180,E1 -5228.14,E2 -5228.14} C_VEL
LIN {X 0,Y 516.504,Z 321.999,A -85,B 0,C 180,E1 -5231.565,E2 -5231.565} C_VEL
LIN {X 0,Y 516.545,Z 314.007,A -85,B 0,C 180,E1 -5234.98,E2 -5234.98} C_VEL
LIN {X 0,Y 516.577,Z 306.397,A -85,B 0,C 180,E1 -5238.234,E2 -5238.234} C_VEL
LIN {X 0,Y 516.617,Z 300.611,A -85,B 0,C 180,E1 -5240.713,E2 -5240.713} C_VEL
LIN {X 0,Y 516.643,Z 294.724,A -85,B 0,C 180,E1 -5243.233,E2 -5243.233} C_VEL
LIN {X 0,Y 516.679,Z 287.785,A -85,B 0,C 180,E1 -5246.136,E2 -5246.136} C_VEL
LIN {X 0,Y 516.805,Z 280.114,A -85,B 0,C 180,E1 -5249.31,E2 -5249.31} C_VEL
LIN {X 0,Y 516.886,Z 280.095,A -85,B 0,C 180,E1 -5252.541,E2 -5252.541} C_VEL
LIN {X 0,Y 516.853,Z 280.105,A -85,B 0,C 180,E1 -5255.327,E2 -5255.327} C_VEL
LIN {X 0,Y 516.871,Z 280.097,A -85,B 0,C 180,E1 -5257.941,E2 -5257.941} C_VEL
LIN {X 0,Y 516.857,Z 280.105,A -85,B 0,C 180,E1 -5260.742,E2 -5260.742} C_VEL
LIN {X 0,Y 516.847,Z 280.107,A -85,B 0,C 180,E1 -5262.833,E2 -5262.833} C_VEL
LIN {X 0,Y 516.887,Z 280.099,A -85,B 0,C 180,E1 -5265.006,E2 -5265.006} C_VEL
LIN {X 0,Y 516.907,Z 280.1,A -85,B 0,C 180,E1 -5268.397,E2 -5268.397} C_VEL
LIN {X 0,Y 516.874,Z 280.098,A -85,B 0,C 180,E1 -5269.466,E2 -5269.466} C_VEL
LIN {X 0,Y 516.213,Z 280.185,A -85,B 0,C 180,E1 -5270.117,E2 -5270.117} C_VEL
LIN {X 0,Y 513.344,Z 280.542,A -85,B 0,C 180,E1 -5271.173,E2 -5271.173} C_VEL
LIN {X 0,Y 510.92,Z 280.844,A -85,B 0,C 180,E1 -5272.024,E2 -5272.024} C_VEL
LIN {X 0,Y 509.889,Z 280.971,A -85,B 0,C 180,E1 -5272.682,E2 -5272.682} C_VEL
LIN {X 0,Y 509.81,Z 280.979,A -85,B 0,C 180,E1 -5272.904,E2 -5272.904} C_VEL
LIN {X 0,Y 509.853,Z 280.977,A -85,B 0,C 180,E1 -5275.795,E2 -5275.795} C_VEL
LIN {X 0,Y 509.839,Z 280.975,A -85,B 0,C 180,E1 -5278.719,E2 -5278.719} C_VEL
LIN {X 0,Y 509.876,Z 280.972,A -85,B 0,C 180,E1 -5281.156,E2 -5281.156} C_VEL
LIN {X 0,Y 509.901,Z 280.971,A -85,B 0,C 180,E1 -5283.828,E2 -5283.828} C_VEL
LIN {X 0,Y 509.826,Z 280.976,A -85,B 0,C 180,E1 -5286.436,E2 -5286.436} C_VEL
LIN {X 0,Y 509.906,Z 280.967,A -85,B 0,C 180,E1 -5289.844,E2 -5289.844} C_VEL
LIN {X 0,Y 509.872,Z 280.974,A -85,B 0,C 180,E1 -5293.174,E2 -5293.174} C_VEL
LIN {X 0,Y 509.852,Z 280.973,A -85,B 0,C 180,E1 -5295.634,E2 -5295.634} C_VEL
LIN {X 0,Y 509.899,Z 280.97,A -85,B 0,C 180,E1 -5298.874,E2 -5298.874} C_VEL
LIN {X 0,Y 509.906,Z 280.969,A -85,B 0,C 180,E1 -5302.078,E2 -5302.078} C_VEL
LIN {X 0,Y 509.956,Z 280.964,A -85,B 0,C 180,E1 -5304.464,E2 -5304.464} C_VEL
LIN {X 0,Y 510.03,Z 280.951,A -85,B 0,C 180,E1 -5307.631,E2 -5307.631} C_VEL
LIN {X 0,Y 510.021,Z 280.959,A -85,B 0,C 180,E1 -5310,E2 -5310} C_VEL
LIN {X 0,Y 510.031,Z 280.951,A -85,B 0,C 180,E1 -5312.369,E2 -5312.369} C_VEL
LIN {X 0,Y 509.957,Z 280.964,A -85,B 0,C 180,E1 -5315.536,E2 -5315.536} C_VEL
LIN {X 0,Y 509.897,Z 280.967,A -85,B 0,C 180,E1 -5318.721,E2 -5318.721} C_VEL
LIN {X 0,Y 509.892,Z 280.969,A -85,B 0,C 180,E1 -5321.932,E2 -5321.932} C_VEL
LIN {X 0,Y 509.882,Z 280.976,A -85,B 0,C 180,E1 -5325.242,E2 -5325.242} C_VEL
LIN {X 0,Y 509.877,Z 280.97,A -85,B 0,C 180,E1 -5328.002,E2 -5328.002} C_VEL
LIN {X 0,Y 509.84,Z 280.98,A -85,B 0,C 180,E1 -5331.002,E2 -5331.002} C_VEL
LIN {X 0,Y 509.826,Z 280.976,A -85,B 0,C 180,E1 -5333.564,E2 -5333.564} C_VEL
LIN {X 0,Y 509.904,Z 280.971,A -85,B 0,C 180,E1 -5336.38,E2 -5336.38} C_VEL
LIN {X 0,Y 509.876,Z 280.972,A -85,B 0,C 180,E1 -5338.844,E2 -5338.844} C_VEL
LIN {X 0,Y 509.817,Z 280.979,A -85,B 0,C 180,E1 -5341.591,E2 -5341.591} C_VEL
LIN {X 0,Y 509.846,Z 280.977,A -85,B 0,C 180,E1 -5344.414,E2 -5344.414} C_VEL
LIN {X 0,Y 509.811,Z 280.98,A -85,B 0,C 180,E1 -5347.342,E2 -5347.342} C_VEL
LIN {X 0,Y 509.83,Z 280.976,A -85,B 0,C 180,E1 -5350.383,E2 -5350.383} C_VEL
LIN {X 0,Y 509.815,Z 280.98,A -85,B 0,C 180,E1 -5353.063,E2 -5353.063} C_VEL
LIN {X 0,Y 509.814,Z 280.98,A -85,B 0,C 180,E1 -5355.795,E2 -5355.795} C_VEL
LIN {X 0,Y 509.837,Z 280.975,A -85,B 0,C 180,E1 -5358.575,E2 -5358.575} C_VEL
LIN {X 0,Y 509.842,Z 280.973,A -85,B 0,C 180,E1 -5361.788,E2 -5361.788} C_VEL
LIN {X 0,Y 509.812,Z 280.982,A -85,B 0,C 180,E1 -5364.622,E2 -5364.622} C_VEL
LIN {X 0,Y 509.852,Z 280.971,A -85,B 0,C 180,E1 -5367.482,E2 -5367.482} C_VEL
LIN {X 0,Y 509.928,Z 281.049,A -85,B 0,C 180,E1 -5369.925,E2 -5369.925} C_VEL
LIN {X 0,Y 509.81,Z 287.459,A -85,B 0,C 180,E1 -5372.942,E2 -5372.942} C_VEL
LIN {X 0,Y 509.676,Z 293.087,A -85,B 0,C 180,E1 -5375.566,E2 -5375.566} C_VEL
LIN {X 0,Y 509.591,Z 298.699,A -85,B 0,C 180,E1 -5378.14,E2 -5378.14} C_VEL
LIN {X 0,Y 509.511,Z 304.247,A -85,B 0,C 180,E1 -5380.669,E2 -5380.669} C_VEL
LIN {X 0,Y 509.405,Z 309.759,A -85,B 0,C 180,E1 -5383.16,E2 -5383.16} C_VEL
LIN {X 0,Y 509.394,Z 315.262,A -85,B 0,C 180,E1 -5385.622,E2 -5385.622} C_VEL
LIN {X 0,Y 509.314,Z 322.569,A -85,B 0,C 180,E1 -5388.862,E2 -5388.862} C_VEL
LIN {X 0,Y 509.294,Z 329.06,A -85,B 0,C 180,E1 -5391.695,E2 -5391.695} C_VEL
LIN {X 0,Y 510.18,Z 337.085,A -85,B 0,C 180,E1 -5392.033,E2 -5392.033} C_VEL
LIN {X 0,Y 510.031,Z 345.494,A -85,B 0,C 180,E1 -5392.479,E2 -5392.479} C_VEL
LIN {X 0,Y 509.883,Z 354.646,A -85,B 0,C 180,E1 -5393.139,E2 -5393.139} C_VEL
LIN {X 0,Y 509.643,Z 362.33,A -85,B 0,C 180,E1 -5393.866,E2 -5393.866} C_VEL
LIN {X 0,Y 509.625,Z 368.827,A -85,B 0,C 180,E1 -5394.66,E2 -5394.66} C_VEL
LIN {X 0,Y 509.536,Z 375.053,A -85,B 0,C 180,E1 -5395.65,E2 -5395.65} C_VEL
LIN {X 0,Y 509.365,Z 380.402,A -85,B 0,C 180,E1 -5396.837,E2 -5396.837} C_VEL
LIN {X 0,Y 509.255,Z 382.916,A -85,B 0,C 180,E1 -5397.628,E2 -5397.628} C_VEL
LIN {X 0,Y 509.203,Z 384.675,A -85,B 0,C 180,E1 -5398.419,E2 -5398.419} C_VEL
LIN {X 0,Y 509.193,Z 385.73,A -85,B 0,C 180,E1 -5399.21,E2 -5399.21} C_VEL
LIN {X 0,Y 509.195,Z 386.142,A -85,B 0,C 180,E1 -5400.001,E2 -5400.001} C_VEL
LIN {X 0,Y 509.2,Z 385.906,A -85,B 0,C 180,E1 -5400.792,E2 -5400.792} C_VEL
LIN {X 0,Y 509.217,Z 385.001,A -85,B 0,C 180,E1 -5401.583,E2 -5401.583} C_VEL
LIN {X 0,Y 509.399,Z 382.302,A -85,B 0,C 180,E1 -5402.769,E2 -5402.769} C_VEL
LIN {X 0,Y 509.525,Z 379.58,A -85,B 0,C 180,E1 -5403.56,E2 -5403.56} C_VEL
LIN {X 0,Y 509.561,Z 374.965,A -85,B 0,C 180,E1 -5404.55,E2 -5404.55} C_VEL
LIN {X 0,Y 509.682,Z 370.122,A -85,B 0,C 180,E1 -5405.342,E2 -5405.342} C_VEL
LIN {X 0,Y 509.786,Z 363.95,A -85,B 0,C 180,E1 -5406.134,E2 -5406.134} C_VEL
LIN {X 0,Y 510.006,Z 356.738,A -85,B 0,C 180,E1 -5406.858,E2 -5406.858} C_VEL
LIN {X 0,Y 510.092,Z 348.785,A -85,B 0,C 180,E1 -5407.482,E2 -5407.482} C_VEL
LIN {X 0,Y 510.287,Z 339.672,A -85,B 0,C 180,E1 -5408.017,E2 -5408.017} C_VEL
LIN {X 0,Y 509.875,Z 332.973,A -85,B 0,C 180,E1 -5408.323,E2 -5408.323} C_VEL
LIN {X 0,Y 509.359,Z 329.941,A -85,B 0,C 180,E1 -5408.456,E2 -5408.456} C_VEL
LIN {X 0,Y 509.477,Z 322.843,A -85,B 0,C 180,E1 -5411.645,E2 -5411.645} C_VEL
LIN {X 0,Y 509.578,Z 315.071,A -85,B 0,C 180,E1 -5415.192,E2 -5415.192} C_VEL
LIN {X 0,Y 509.691,Z 309.214,A -85,B 0,C 180,E1 -5417.931,E2 -5417.931} C_VEL
LIN {X 0,Y 509.82,Z 302.623,A -85,B 0,C 180,E1 -5421.004,E2 -5421.004} C_VEL
LIN {X 0,Y 509.96,Z 295.353,A -85,B 0,C 180,E1 -5424.422,E2 -5424.422} C_VEL
LIN {X 0,Y 510.078,Z 289.85,A -85,B 0,C 180,E1 -5427.045,E2 -5427.045} C_VEL
LIN {X 0,Y 510.199,Z 284.167,A -85,B 0,C 180,E1 -5429.793,E2 -5429.793} C_VEL
LIN {X 0,Y 509.864,Z 280.979,A -85,B 0,C 180,E1 -5431.445,E2 -5431.445} C_VEL
LIN {X 0,Y 509.853,Z 280.979,A -85,B 0,C 180,E1 -5434.414,E2 -5434.414} C_VEL
LIN {X 0,Y 509.822,Z 280.982,A -85,B 0,C 180,E1 -5437.341,E2 -5437.341} C_VEL
LIN {X 0,Y 509.843,Z 280.979,A -85,B 0,C 180,E1 -5440.383,E2 -5440.383} C_VEL
LIN {X 0,Y 509.828,Z 280.982,A -85,B 0,C 180,E1 -5443.062,E2 -5443.062} C_VEL
LIN {X 0,Y 509.827,Z 280.98,A -85,B 0,C 180,E1 -5445.794,E2 -5445.794} C_VEL
LIN {X 0,Y 509.86,Z 280.978,A -85,B 0,C 180,E1 -5448.575,E2 -5448.575} C_VEL
LIN {X 0,Y 509.855,Z 280.979,A -85,B 0,C 180,E1 -5451.787,E2 -5451.787} C_VEL
LIN {X 0,Y 509.834,Z 280.982,A -85,B 0,C 180,E1 -5454.622,E2 -5454.622} C_VEL
LIN {X 0,Y 509.854,Z 280.981,A -85,B 0,C 180,E1 -5457.714,E2 -5457.714} C_VEL
LIN {X 0,Y 509.857,Z 281.151,A -85,B 0,C 180,E1 -5457.948,E2 -5457.948} C_VEL
LIN {X 0,Y 511.848,Z 289.806,A -85,B 0,C 180,E1 -5460.376,E2 -5460.376} C_VEL
LIN {X 0,Y 512.647,Z 293.591,A -85,B 0,C 180,E1 -5461.33,E2 -5461.33} C_VEL
LIN {X 0,Y 512.53,Z 298.464,A -85,B 0,C 180,E1 -5462.432,E2 -5462.432} C_VEL
LIN {X 0,Y 511.711,Z 310.862,A -85,B 0,C 180,E1 -5465.022,E2 -5465.022} C_VEL
LIN {X 0,Y 511.079,Z 323.878,A -85,B 0,C 180,E1 -5467.567,E2 -5467.567} C_VEL
LIN {X 0,Y 510.683,Z 336.156,A -85,B 0,C 180,E1 -5469.876,E2 -5469.876} C_VEL
LIN {X 0,Y 510.262,Z 352.12,A -85,B 0,C 180,E1 -5472.775,E2 -5472.775} C_VEL
LIN {X 0,Y 509.913,Z 370.607,A -85,B 0,C 180,E1 -5476.017,E2 -5476.017} C_VEL
LIN {X 0,Y 511.27,Z 383.9,A -85,B 0,C 180,E1 -5476.334,E2 -5476.334} C_VEL
LIN {X 0,Y 511.036,Z 397.566,A -85,B 0,C 180,E1 -5476.783,E2 -5476.783} C_VEL
LIN {X 0,Y 510.742,Z 410.124,A -85,B 0,C 180,E1 -5477.371,E2 -5477.371} C_VEL
LIN {X 0,Y 510.515,Z 421.653,A -85,B 0,C 180,E1 -5478.083,E2 -5478.083} C_VEL
LIN {X 0,Y 510.177,Z 432,A -85,B 0,C 180,E1 -5478.88,E2 -5478.88} C_VEL
LIN {X 0,Y 509.894,Z 442.429,A -85,B 0,C 180,E1 -5479.878,E2 -5479.878} C_VEL
LIN {X 0,Y 509.681,Z 450.896,A -85,B 0,C 180,E1 -5480.876,E2 -5480.876} C_VEL
LIN {X 0,Y 509.514,Z 459.179,A -85,B 0,C 180,E1 -5482.072,E2 -5482.072} C_VEL
LIN {X 0,Y 509.38,Z 466.029,A -85,B 0,C 180,E1 -5483.305,E2 -5483.305} C_VEL
LIN {X 0,Y 509.339,Z 471.105,A -85,B 0,C 180,E1 -5484.457,E2 -5484.457} C_VEL
LIN {X 0,Y 509.274,Z 475.189,A -85,B 0,C 180,E1 -5485.647,E2 -5485.647} C_VEL
LIN {X 0,Y 509.259,Z 478.206,A -85,B 0,C 180,E1 -5486.836,E2 -5486.836} C_VEL
LIN {X 0,Y 509.192,Z 479.639,A -85,B 0,C 180,E1 -5487.627,E2 -5487.627} C_VEL
LIN {X 0,Y 509.11,Z 481.283,A -85,B 0,C 180,E1 -5489.209,E2 -5489.209} C_VEL
LIN {X 0,Y 509.108,Z 481.513,A -85,B 0,C 180,E1 -5490,E2 -5490} C_VEL
LIN {X 0,Y 509.109,Z 481.296,A -85,B 0,C 180,E1 -5490.791,E2 -5490.791} C_VEL
LIN {X 0,Y 509.192,Z 479.677,A -85,B 0,C 180,E1 -5492.373,E2 -5492.373} C_VEL
LIN {X 0,Y 509.259,Z 478.256,A -85,B 0,C 180,E1 -5493.164,E2 -5493.164} C_VEL
LIN {X 0,Y 509.273,Z 475.267,A -85,B 0,C 180,E1 -5494.353,E2 -5494.353} C_VEL
LIN {X 0,Y 509.339,Z 471.215,A -85,B 0,C 180,E1 -5495.543,E2 -5495.543} C_VEL
LIN {X 0,Y 509.405,Z 465.408,A -85,B 0,C 180,E1 -5496.844,E2 -5496.844} C_VEL
LIN {X 0,Y 509.528,Z 458.112,A -85,B 0,C 180,E1 -5498.128,E2 -5498.128} C_VEL
LIN {X 0,Y 509.727,Z 449.609,A -85,B 0,C 180,E1 -5499.323,E2 -5499.323} C_VEL
LIN {X 0,Y 509.973,Z 440.827,A -85,B 0,C 180,E1 -5500.321,E2 -5500.321} C_VEL
LIN {X 0,Y 510.304,Z 430.009,A -85,B 0,C 180,E1 -5501.318,E2 -5501.318} C_VEL
LIN {X 0,Y 510.587,Z 418.574,A -85,B 0,C 180,E1 -5502.158,E2 -5502.158} C_VEL
LIN {X 0,Y 510.853,Z 407.079,A -85,B 0,C 180,E1 -5502.817,E2 -5502.817} C_VEL
LIN {X 0,Y 511.148,Z 394.438,A -85,B 0,C 180,E1 -5503.366,E2 -5503.366} C_VEL
LIN {X 0,Y 511.242,Z 382.066,A -85,B 0,C 180,E1 -5503.743,E2 -5503.743} C_VEL
LIN {X 0,Y 509.91,Z 370.821,A -85,B 0,C 180,E1 -5504.008,E2 -5504.008} C_VEL
LIN {X 0,Y 510.252,Z 353.923,A -85,B 0,C 180,E1 -5507.019,E2 -5507.019} C_VEL
LIN {X 0,Y 510.825,Z 335.285,A -85,B 0,C 180,E1 -5510.413,E2 -5510.413} C_VEL
LIN {X 0,Y 511.517,Z 316.615,A -85,B 0,C 180,E1 -5513.911,E2 -5513.911} C_VEL
LIN {X 0,Y 512.193,Z 301.006,A -85,B 0,C 180,E1 -5516.924,E2 -5516.924} C_VEL
LIN {X 0,Y 512.507,Z 294.366,A -85,B 0,C 180,E1 -5518.236,E2 -5518.236} C_VEL
LIN {X 0,Y 511.332,Z 287.752,A -85,B 0,C 180,E1 -5519.657,E2 -5519.657} C_VEL
LIN {X 0,Y 509.849,Z 280.978,A -85,B 0,C 180,E1 -5521.206,E2 -5521.206} C_VEL
LIN {X 0,Y 509.847,Z 280.98,A -85,B 0,C 180,E1 -5524.2,E2 -5524.2} C_VEL
LIN {X 0,Y 509.821,Z 280.983,A -85,B 0,C 180,E1 -5527.341,E2 -5527.341} C_VEL
LIN {X 0,Y 509.843,Z 280.979,A -85,B 0,C 180,E1 -5530.382,E2 -5530.382} C_VEL
LIN {X 0,Y 509.828,Z 280.98,A -85,B 0,C 180,E1 -5533.062,E2 -5533.062} C_VEL
LIN {X 0,Y 509.836,Z 280.98,A -85,B 0,C 180,E1 -5535.792,E2 -5535.792} C_VEL
LIN {X 0,Y 509.86,Z 280.976,A -85,B 0,C 180,E1 -5538.574,E2 -5538.574} C_VEL
LIN {X 0,Y 509.857,Z 280.977,A -85,B 0,C 180,E1 -5541.786,E2 -5541.786} C_VEL
LIN {X 0,Y 509.835,Z 280.981,A -85,B 0,C 180,E1 -5544.621,E2 -5544.621} C_VEL
LIN {X 0,Y 509.865,Z 280.979,A -85,B 0,C 180,E1 -5547.48,E2 -5547.48} C_VEL
LIN {X 0,Y 509.798,Z 280.985,A -85,B 0,C 180,E1 -5550.286,E2 -5550.286} C_VEL
LIN {X 0,Y 509.583,Z 281.034,A -85,B 0,C 180,E1 -5551.884,E2 -5551.884} C_VEL
LIN {X 0,Y 509.554,Z 290.17,A -85,B 0,C 180,E1 -5555.123,E2 -5555.123} C_VEL
LIN {X 0,Y 509.568,Z 296.565,A -85,B 0,C 180,E1 -5557.529,E2 -5557.529} C_VEL
LIN {X 0,Y 509.584,Z 303.414,A -85,B 0,C 180,E1 -5560.25,E2 -5560.25} C_VEL
LIN {X 0,Y 509.502,Z 310.608,A -85,B 0,C 180,E1 -5563.161,E2 -5563.161} C_VEL
LIN {X 0,Y 509.52,Z 316.542,A -85,B 0,C 180,E1 -5565.623,E2 -5565.623} C_VEL
LIN {X 0,Y 509.512,Z 324.219,A -85,B 0,C 180,E1 -5568.865,E2 -5568.865} C_VEL
LIN {X 0,Y 509.487,Z 331.316,A -85,B 0,C 180,E1 -5571.871,E2 -5571.871} C_VEL
LIN {X 0,Y 510.095,Z 337.839,A -85,B 0,C 180,E1 -5572.13,E2 -5572.13} C_VEL
LIN {X 0,Y 509.961,Z 346.423,A -85,B 0,C 180,E1 -5572.576,E2 -5572.576} C_VEL
LIN {X 0,Y 509.889,Z 354.45,A -85,B 0,C 180,E1 -5573.131,E2 -5573.131} C_VEL
LIN {X 0,Y 509.643,Z 362.366,A -85,B 0,C 180,E1 -5573.864,E2 -5573.864} C_VEL
LIN {X 0,Y 509.678,Z 369.001,A -85,B 0,C 180,E1 -5574.658,E2 -5574.658} C_VEL
LIN {X 0,Y 509.555,Z 374.085,A -85,B 0,C 180,E1 -5575.45,E2 -5575.45} C_VEL
LIN {X 0,Y 509.523,Z 378.998,A -85,B 0,C 180,E1 -5576.44,E2 -5576.44} C_VEL
LIN {X 0,Y 509.397,Z 381.87,A -85,B 0,C 180,E1 -5577.231,E2 -5577.231} C_VEL
LIN {X 0,Y 509.206,Z 384.709,A -85,B 0,C 180,E1 -5578.417,E2 -5578.417} C_VEL
LIN {X 0,Y 509.189,Z 385.742,A -85,B 0,C 180,E1 -5579.208,E2 -5579.208} C_VEL
LIN {X 0,Y 509.184,Z 386.1,A -85,B 0,C 180,E1 -5579.999,E2 -5579.999} C_VEL
LIN {X 0,Y 509.184,Z 385.789,A -85,B 0,C 180,E1 -5580.79,E2 -5580.79} C_VEL
LIN {X 0,Y 509.199,Z 384.805,A -85,B 0,C 180,E1 -5581.581,E2 -5581.581} C_VEL
LIN {X 0,Y 509.394,Z 381.98,A -85,B 0,C 180,E1 -5582.767,E2 -5582.767} C_VEL
LIN {X 0,Y 509.411,Z 379.191,A -85,B 0,C 180,E1 -5583.558,E2 -5583.558} C_VEL
LIN {X 0,Y 509.548,Z 374.38,A -85,B 0,C 180,E1 -5584.548,E2 -5584.548} C_VEL
LIN {X 0,Y 509.598,Z 369.357,A -85,B 0,C 180,E1 -5585.34,E2 -5585.34} C_VEL
LIN {X 0,Y 509.621,Z 362.939,A -85,B 0,C 180,E1 -5586.134,E2 -5586.134} C_VEL
LIN {X 0,Y 509.826,Z 356.09,A -85,B 0,C 180,E1 -5586.789,E2 -5586.789} C_VEL
LIN {X 0,Y 509.944,Z 347.611,A -85,B 0,C 180,E1 -5587.423,E2 -5587.423} C_VEL
LIN {X 0,Y 510.002,Z 338.348,A -85,B 0,C 180,E1 -5587.92,E2 -5587.92} C_VEL
LIN {X 0,Y 509.797,Z 333.443,A -85,B 0,C 180,E1 -5588.122,E2 -5588.122} C_VEL
LIN {X 0,Y 509.366,Z 330.58,A -85,B 0,C 180,E1 -5588.254,E2 -5588.254} C_VEL
LIN {X 0,Y 509.419,Z 323.807,A -85,B 0,C 180,E1 -5591.135,E2 -5591.135} C_VEL
LIN {X 0,Y 509.454,Z 316.217,A -85,B 0,C 180,E1 -5594.376,E2 -5594.376} C_VEL
LIN {X 0,Y 509.472,Z 310.478,A -85,B 0,C 180,E1 -5596.838,E2 -5596.838} C_VEL
LIN {X 0,Y 509.538,Z 304.686,A -85,B 0,C 180,E1 -5599.33,E2 -5599.33} C_VEL
LIN {X 0,Y 509.568,Z 298.761,A -85,B 0,C 180,E1 -5601.861,E2 -5601.861} C_VEL
LIN {X 0,Y 509.622,Z 292.602,A -85,B 0,C 180,E1 -5604.469,E2 -5604.469} C_VEL
LIN {X 0,Y 509.677,Z 285.311,A -85,B 0,C 180,E1 -5607.511,E2 -5607.511} C_VEL
LIN {X 0,Y 509.751,Z 280.992,A -85,B 0,C 180,E1 -5609.302,E2 -5609.302} C_VEL
LIN {X 0,Y 509.792,Z 280.984,A -85,B 0,C 180,E1 -5611.591,E2 -5611.591} C_VEL
LIN {X 0,Y 509.828,Z 280.975,A -85,B 0,C 180,E1 -5614.414,E2 -5614.414} C_VEL
LIN {X 0,Y 509.801,Z 280.982,A -85,B 0,C 180,E1 -5617.34,E2 -5617.34} C_VEL
LIN {X 0,Y 509.811,Z 280.98,A -85,B 0,C 180,E1 -5620.383,E2 -5620.383} C_VEL
LIN {X 0,Y 509.793,Z 280.983,A -85,B 0,C 180,E1 -5623.058,E2 -5623.058} C_VEL
LIN {X 0,Y 509.814,Z 280.978,A -85,B 0,C 180,E1 -5625.792,E2 -5625.792} C_VEL
LIN {X 0,Y 509.849,Z 280.979,A -85,B 0,C 180,E1 -5628.574,E2 -5628.574} C_VEL
LIN {X 0,Y 509.843,Z 280.977,A -85,B 0,C 180,E1 -5631.785,E2 -5631.785} C_VEL
LIN {X 0,Y 509.81,Z 280.979,A -85,B 0,C 180,E1 -5632.904,E2 -5632.904} C_VEL
LIN {X 0,Y 509.157,Z 281.063,A -85,B 0,C 180,E1 -5633.564,E2 -5633.564} C_VEL
LIN {X 0,Y 506.31,Z 281.417,A -85,B 0,C 180,E1 -5634.636,E2 -5634.636} C_VEL
LIN {X 0,Y 503.9,Z 281.718,A -85,B 0,C 180,E1 -5635.499,E2 -5635.499} C_VEL
LIN {X 0,Y 502.872,Z 281.848,A -85,B 0,C 180,E1 -5636.165,E2 -5636.165} C_VEL
LIN {X 0,Y 502.792,Z 281.853,A -85,B 0,C 180,E1 -5636.391,E2 -5636.391} C_VEL
LIN {X 0,Y 502.81,Z 281.855,A -85,B 0,C 180,E1 -5639.789,E2 -5639.789} C_VEL
LIN {X 0,Y 502.826,Z 281.849,A -85,B 0,C 180,E1 -5642.533,E2 -5642.533} C_VEL
LIN {X 0,Y 502.818,Z 281.854,A -85,B 0,C 180,E1 -5645.298,E2 -5645.298} C_VEL
LIN {X 0,Y 502.783,Z 281.855,A -85,B 0,C 180,E1 -5647.826,E2 -5647.826} C_VEL
LIN {X 0,Y 502.815,Z 281.85,A -85,B 0,C 180,E1 -5650.4,E2 -5650.4} C_VEL
LIN {X 0,Y 502.822,Z 281.854,A -85,B 0,C 180,E1 -5652.931,E2 -5652.931} C_VEL
LIN {X 0,Y 502.833,Z 281.848,A -85,B 0,C 180,E1 -5655.429,E2 -5655.429} C_VEL
LIN {X 0,Y 502.864,Z 281.848,A -85,B 0,C 180,E1 -5658.716,E2 -5658.716} C_VEL
LIN {X 0,Y 502.866,Z 281.845,A -85,B 0,C 180,E1 -5661.966,E2 -5661.966} C_VEL
LIN {X 0,Y 502.909,Z 281.843,A -85,B 0,C 180,E1 -5664.386,E2 -5664.386} C_VEL
LIN {X 0,Y 502.998,Z 281.827,A -85,B 0,C 180,E1 -5667.598,E2 -5667.598} C_VEL
LIN {X 0,Y 502.99,Z 281.834,A -85,B 0,C 180,E1 -5670,E2 -5670} C_VEL
LIN {X 0,Y 502.998,Z 281.827,A -85,B 0,C 180,E1 -5672.402,E2 -5672.402} C_VEL
LIN {X 0,Y 502.91,Z 281.843,A -85,B 0,C 180,E1 -5675.614,E2 -5675.614} C_VEL
LIN {X 0,Y 502.856,Z 281.845,A -85,B 0,C 180,E1 -5678.844,E2 -5678.844} C_VEL
LIN {X 0,Y 502.833,Z 281.847,A -85,B 0,C 180,E1 -5682.102,E2 -5682.102} C_VEL
LIN {X 0,Y 502.836,Z 281.851,A -85,B 0,C 180,E1 -5685.4,E2 -5685.4} C_VEL
LIN {X 0,Y 502.835,Z 281.847,A -85,B 0,C 180,E1 -5688.123,E2 -5688.123} C_VEL
LIN {X 0,Y 502.818,Z 281.853,A -85,B 0,C 180,E1 -5690.537,E2 -5690.537} C_VEL
LIN {X 0,Y 502.786,Z 281.857,A -85,B 0,C 180,E1 -5693.041,E2 -5693.041} C_VEL
LIN {X 0,Y 502.831,Z 281.848,A -85,B 0,C 180,E1 -5695.676,E2 -5695.676} C_VEL
LIN {X 0,Y 502.833,Z 281.852,A -85,B 0,C 180,E1 -5698.373,E2 -5698.373} C_VEL
LIN {X 0,Y 502.788,Z 281.854,A -85,B 0,C 180,E1 -5701.501,E2 -5701.501} C_VEL
LIN {X 0,Y 502.798,Z 281.855,A -85,B 0,C 180,E1 -5704.446,E2 -5704.446} C_VEL
LIN {X 0,Y 502.773,Z 281.856,A -85,B 0,C 180,E1 -5707.179,E2 -5707.179} C_VEL
LIN {X 0,Y 502.78,Z 281.857,A -85,B 0,C 180,E1 -5710.016,E2 -5710.016} C_VEL
LIN {X 0,Y 502.795,Z 281.853,A -85,B 0,C 180,E1 -5712.2,E2 -5712.2} C_VEL
LIN {X 0,Y 502.778,Z 281.859,A -85,B 0,C 180,E1 -5715.471,E2 -5715.471} C_VEL
LIN {X 0,Y 502.788,Z 281.853,A -85,B 0,C 180,E1 -5717.862,E2 -5717.862} C_VEL
LIN {X 0,Y 502.786,Z 281.86,A -85,B 0,C 180,E1 -5721.024,E2 -5721.024} C_VEL
LIN {X 0,Y 502.759,Z 281.856,A -85,B 0,C 180,E1 -5724.172,E2 -5724.172} C_VEL
LIN {X 0,Y 502.797,Z 281.854,A -85,B 0,C 180,E1 -5727,E2 -5727} C_VEL
LIN {X 0,Y 502.888,Z 281.911,A -85,B 0,C 180,E1 -5729.876,E2 -5729.876} C_VEL
LIN {X 0,Y 502.779,Z 287.483,A -85,B 0,C 180,E1 -5732.532,E2 -5732.532} C_VEL
LIN {X 0,Y 502.644,Z 293.497,A -85,B 0,C 180,E1 -5735.345,E2 -5735.345} C_VEL
LIN {X 0,Y 502.549,Z 298.826,A -85,B 0,C 180,E1 -5737.817,E2 -5737.817} C_VEL
LIN {X 0,Y 502.457,Z 304.405,A -85,B 0,C 180,E1 -5740.387,E2 -5740.387} C_VEL
LIN {X 0,Y 502.358,Z 309.968,A -85,B 0,C 180,E1 -5742.916,E2 -5742.916} C_VEL
LIN {X 0,Y 502.337,Z 315.496,A -85,B 0,C 180,E1 -5745.415,E2 -5745.415} C_VEL
LIN {X 0,Y 502.269,Z 322.845,A -85,B 0,C 180,E1 -5748.704,E2 -5748.704} C_VEL
LIN {X 0,Y 502.237,Z 329.319,A -85,B 0,C 180,E1 -5751.552,E2 -5751.552} C_VEL
LIN {X 0,Y 503.203,Z 337.885,A -85,B 0,C 180,E1 -5751.922,E2 -5751.922} C_VEL
LIN {X 0,Y 503.046,Z 346.177,A -85,B 0,C 180,E1 -5752.374,E2 -5752.374} C_VEL
LIN {X 0,Y 502.89,Z 355.28,A -85,B 0,C 180,E1 -5753.043,E2 -5753.043} C_VEL
LIN {X 0,Y 502.614,Z 362.95,A -85,B 0,C 180,E1 -5753.78,E2 -5753.78} C_VEL
LIN {X 0,Y 502.598,Z 369.443,A -85,B 0,C 180,E1 -5754.585,E2 -5754.585} C_VEL
LIN {X 0,Y 502.502,Z 375.664,A -85,B 0,C 180,E1 -5755.589,E2 -5755.589} C_VEL
LIN {X 0,Y 502.364,Z 379.448,A -85,B 0,C 180,E1 -5756.392,E2 -5756.392} C_VEL
LIN {X 0,Y 502.191,Z 383.554,A -85,B 0,C 180,E1 -5757.595,E2 -5757.595} C_VEL
LIN {X 0,Y 502.137,Z 385.329,A -85,B 0,C 180,E1 -5758.397,E2 -5758.397} C_VEL
LIN {X 0,Y 502.127,Z 386.405,A -85,B 0,C 180,E1 -5759.199,E2 -5759.199} C_VEL
LIN {X 0,Y 502.128,Z 386.825,A -85,B 0,C 180,E1 -5760.001,E2 -5760.001} C_VEL
LIN {X 0,Y 502.134,Z 386.59,A -85,B 0,C 180,E1 -5760.803,E2 -5760.803} C_VEL
LIN {X 0,Y 502.154,Z 385.685,A -85,B 0,C 180,E1 -5761.605,E2 -5761.605} C_VEL
LIN {X 0,Y 502.355,Z 382.999,A -85,B 0,C 180,E1 -5762.808,E2 -5762.808} C_VEL
LIN {X 0,Y 502.493,Z 380.275,A -85,B 0,C 180,E1 -5763.609,E2 -5763.609} C_VEL
LIN {X 0,Y 502.532,Z 375.677,A -85,B 0,C 180,E1 -5764.613,E2 -5764.613} C_VEL
LIN {X 0,Y 502.666,Z 370.838,A -85,B 0,C 180,E1 -5765.416,E2 -5765.416} C_VEL
LIN {X 0,Y 502.774,Z 364.7,A -85,B 0,C 180,E1 -5766.22,E2 -5766.22} C_VEL
LIN {X 0,Y 503.018,Z 357.674,A -85,B 0,C 180,E1 -5766.943,E2 -5766.943} C_VEL
LIN {X 0,Y 503.12,Z 349.693,A -85,B 0,C 180,E1 -5767.586,E2 -5767.586} C_VEL
LIN {X 0,Y 503.333,Z 339.77,A -85,B 0,C 180,E1 -5768.179,E2 -5768.179} C_VEL
LIN {X 0,Y 502.995,Z 334.318,A -85,B 0,C 180,E1 -5768.437,E2 -5768.437} C_VEL
LIN {X 0,Y 502.333,Z 330.354,A -85,B 0,C 180,E1 -5768.626,E2 -5768.626} C_VEL
LIN {X 0,Y 502.434,Z 323.53,A -85,B 0,C 180,E1 -5771.718,E2 -5771.718} C_VEL
LIN {X 0,Y 502.541,Z 315.545,A -85,B 0,C 180,E1 -5775.41,E2 -5775.41} C_VEL
LIN {X 0,Y 502.654,Z 309.888,A -85,B 0,C 180,E1 -5778.054,E2 -5778.054} C_VEL
LIN {X 0,Y 502.772,Z 304.708,A -85,B 0,C 180,E1 -5780.518,E2 -5780.518} C_VEL
LIN {X 0,Y 502.91,Z 297.6,A -85,B 0,C 180,E1 -5783.909,E2 -5783.909} C_VEL
LIN {X 0,Y 503.07,Z 292.037,A -85,B 0,C 180,E1 -5786.607,E2 -5786.607} C_VEL
LIN {X 0,Y 503.218,Z 286.629,A -85,B 0,C 180,E1 -5789.264,E2 -5789.264} C_VEL
LIN {X 0,Y 502.875,Z 282.249,A -85,B 0,C 180,E1 -5791.513,E2 -5791.513} C_VEL
LIN {X 0,Y 502.804,Z 281.858,A -85,B 0,C 180,E1 -5791.757,E2 -5791.757} C_VEL
LIN {X 0,Y 502.806,Z 281.857,A -85,B 0,C 180,E1 -5794.444,E2 -5794.444} C_VEL
LIN {X 0,Y 502.783,Z 281.859,A -85,B 0,C 180,E1 -5797.178,E2 -5797.178} C_VEL
LIN {X 0,Y 502.793,Z 281.859,A -85,B 0,C 180,E1 -5800.016,E2 -5800.016} C_VEL
LIN {X 0,Y 502.808,Z 281.856,A -85,B 0,C 180,E1 -5802.2,E2 -5802.2} C_VEL
LIN {X 0,Y 502.791,Z 281.858,A -85,B 0,C 180,E1 -5805.47,E2 -5805.47} C_VEL
LIN {X 0,Y 502.825,Z 281.854,A -85,B 0,C 180,E1 -5808.934,E2 -5808.934} C_VEL
LIN {X 0,Y 502.798,Z 281.857,A -85,B 0,C 180,E1 -5812.046,E2 -5812.046} C_VEL
LIN {X 0,Y 502.804,Z 281.858,A -85,B 0,C 180,E1 -5815.034,E2 -5815.034} C_VEL
LIN {X 0,Y 502.845,Z 281.993,A -85,B 0,C 180,E1 -5817.446,E2 -5817.446} C_VEL
LIN {X 0,Y 504.756,Z 290.333,A -85,B 0,C 180,E1 -5819.917,E2 -5819.917} C_VEL
LIN {X 0,Y 505.88,Z 296.307,A -85,B 0,C 180,E1 -5821.47,E2 -5821.47} C_VEL
LIN {X 0,Y 505.178,Z 306.743,A -85,B 0,C 180,E1 -5823.787,E2 -5823.787} C_VEL
LIN {X 0,Y 504.239,Z 321.985,A -85,B 0,C 180,E1 -5826.912,E2 -5826.912} C_VEL
LIN {X 0,Y 503.679,Z 336.971,A -85,B 0,C 180,E1 -5829.797,E2 -5829.797} C_VEL
LIN {X 0,Y 503.216,Z 352.826,A -85,B 0,C 180,E1 -5832.736,E2 -5832.736} C_VEL
LIN {X 0,Y 502.837,Z 370.299,A -85,B 0,C 180,E1 -5835.868,E2 -5835.868} C_VEL
LIN {X 0,Y 504.278,Z 384.678,A -85,B 0,C 180,E1 -5836.218,E2 -5836.218} C_VEL
LIN {X 0,Y 504.055,Z 397.324,A -85,B 0,C 180,E1 -5836.648,E2 -5836.648} C_VEL
LIN {X 0,Y 503.716,Z 409.127,A -85,B 0,C 180,E1 -5837.206,E2 -5837.206} C_VEL
LIN {X 0,Y 503.491,Z 420.558,A -85,B 0,C 180,E1 -5837.914,E2 -5837.914} C_VEL
LIN {X 0,Y 503.098,Z 432.195,A -85,B 0,C 180,E1 -5838.824,E2 -5838.824} C_VEL
LIN {X 0,Y 502.856,Z 441.539,A -85,B 0,C 180,E1 -5839.735,E2 -5839.735} C_VEL
LIN {X 0,Y 502.621,Z 450.058,A -85,B 0,C 180,E1 -5840.747,E2 -5840.747} C_VEL
LIN {X 0,Y 502.433,Z 458.385,A -85,B 0,C 180,E1 -5841.959,E2 -5841.959} C_VEL
LIN {X 0,Y 502.317,Z 465.28,A -85,B 0,C 180,E1 -5843.21,E2 -5843.21} C_VEL
LIN {X 0,Y 502.274,Z 470.385,A -85,B 0,C 180,E1 -5844.379,E2 -5844.379} C_VEL
LIN {X 0,Y 502.184,Z 474.491,A -85,B 0,C 180,E1 -5845.585,E2 -5845.585} C_VEL
LIN {X 0,Y 502.207,Z 477.528,A -85,B 0,C 180,E1 -5846.791,E2 -5846.791} C_VEL
LIN {X 0,Y 502.125,Z 478.97,A -85,B 0,C 180,E1 -5847.593,E2 -5847.593} C_VEL
LIN {X 0,Y 502.039,Z 480.627,A -85,B 0,C 180,E1 -5849.198,E2 -5849.198} C_VEL
LIN {X 0,Y 502.038,Z 480.86,A -85,B 0,C 180,E1 -5850,E2 -5850} C_VEL
LIN {X 0,Y 502.038,Z 480.644,A -85,B 0,C 180,E1 -5850.802,E2 -5850.802} C_VEL
LIN {X 0,Y 502.125,Z 479.027,A -85,B 0,C 180,E1 -5852.407,E2 -5852.407} C_VEL
LIN {X 0,Y 502.207,Z 477.602,A -85,B 0,C 180,E1 -5853.209,E2 -5853.209} C_VEL
LIN {X 0,Y 502.183,Z 474.603,A -85,B 0,C 180,E1 -5854.415,E2 -5854.415} C_VEL
LIN {X 0,Y 502.275,Z 470.539,A -85,B 0,C 180,E1 -5855.621,E2 -5855.621} C_VEL
LIN {X 0,Y 502.334,Z 464.351,A -85,B 0,C 180,E1 -5857.012,E2 -5857.012} C_VEL
LIN {X 0,Y 502.477,Z 457.392,A -85,B 0,C 180,E1 -5858.243,E2 -5858.243} C_VEL
LIN {X 0,Y 502.621,Z 450.383,A -85,B 0,C 180,E1 -5859.253,E2 -5859.253} C_VEL
LIN {X 0,Y 502.861,Z 441.934,A -85,B 0,C 180,E1 -5860.265,E2 -5860.265} C_VEL
LIN {X 0,Y 503.146,Z 432.684,A -85,B 0,C 180,E1 -5861.175,E2 -5861.175} C_VEL
LIN {X 0,Y 503.517,Z 421.15,A -85,B 0,C 180,E1 -5862.085,E2 -5862.085} C_VEL
LIN {X 0,Y 503.785,Z 409.844,A -85,B 0,C 180,E1 -5862.794,E2 -5862.794} C_VEL
LIN {X 0,Y 504.071,Z 398.297,A -85,B 0,C 180,E1 -5863.351,E2 -5863.351} C_VEL
LIN {X 0,Y 504.325,Z 385.038,A -85,B 0,C 180,E1 -5863.807,E2 -5863.807} C_VEL
LIN {X 0,Y 503.15,Z 373.272,A -85,B 0,C 180,E1 -5864.097,E2 -5864.097} C_VEL
LIN {X 0,Y 502.859,Z 370.634,A -85,B 0,C 180,E1 -5864.157,E2 -5864.157} C_VEL
LIN {X 0,Y 503.203,Z 354.702,A -85,B 0,C 180,E1 -5867.056,E2 -5867.056} C_VEL
LIN {X 0,Y 503.817,Z 336.623,A -85,B 0,C 180,E1 -5870.41,E2 -5870.41} C_VEL
LIN {X 0,Y 504.522,Z 318.686,A -85,B 0,C 180,E1 -5873.827,E2 -5873.827} C_VEL
LIN {X 0,Y 505.252,Z 303.662,A -85,B 0,C 180,E1 -5876.772,E2 -5876.772} C_VEL
LIN {X 0,Y 505.551,Z 295.061,A -85,B 0,C 180,E1 -5878.508,E2 -5878.508} C_VEL
LIN {X 0,Y 503.642,Z 285.515,A -85,B 0,C 180,E1 -5880.619,E2 -5880.619} C_VEL
LIN {X 0,Y 502.798,Z 281.856,A -85,B 0,C 180,E1 -5881.498,E2 -5881.498} C_VEL
LIN {X 0,Y 502.794,Z 281.858,A -85,B 0,C 180,E1 -5883.995,E2 -5883.995} C_VEL
LIN {X 0,Y 502.782,Z 281.859,A -85,B 0,C 180,E1 -5887.177,E2 -5887.177} C_VEL
LIN {X 0,Y 502.793,Z 281.857,A -85,B 0,C 180,E1 -5890.015,E2 -5890.015} C_VEL
LIN {X 0,Y 502.808,Z 281.855,A -85,B 0,C 180,E1 -5892.199,E2 -5892.199} C_VEL
LIN {X 0,Y 502.806,Z 281.855,A -85,B 0,C 180,E1 -5895.468,E2 -5895.468} C_VEL
LIN {X 0,Y 502.825,Z 281.853,A -85,B 0,C 180,E1 -5898.934,E2 -5898.934} C_VEL
LIN {X 0,Y 502.799,Z 281.857,A -85,B 0,C 180,E1 -5902.046,E2 -5902.046} C_VEL
LIN {X 0,Y 502.801,Z 281.856,A -85,B 0,C 180,E1 -5905.034,E2 -5905.034} C_VEL
LIN {X 0,Y 502.788,Z 281.861,A -85,B 0,C 180,E1 -5907.915,E2 -5907.915} C_VEL
LIN {X 0,Y 502.705,Z 281.87,A -85,B 0,C 180,E1 -5910.704,E2 -5910.704} C_VEL
LIN {X 0,Y 502.54,Z 282.019,A -85,B 0,C 180,E1 -5911.898,E2 -5911.898} C_VEL
LIN {X 0,Y 502.51,Z 290.057,A -85,B 0,C 180,E1 -5914.749,E2 -5914.749} C_VEL
LIN {X 0,Y 502.548,Z 297.037,A -85,B 0,C 180,E1 -5917.368,E2 -5917.368} C_VEL
LIN {X 0,Y 502.528,Z 302.661,A -85,B 0,C 180,E1 -5919.557,E2 -5919.557} C_VEL
LIN {X 0,Y 502.484,Z 309.783,A -85,B 0,C 180,E1 -5922.499,E2 -5922.499} C_VEL
LIN {X 0,Y 502.486,Z 316.974,A -85,B 0,C 180,E1 -5925.418,E2 -5925.418} C_VEL
LIN {X 0,Y 502.487,Z 324.775,A -85,B 0,C 180,E1 -5928.707,E2 -5928.707} C_VEL
LIN {X 0,Y 502.449,Z 331.944,A -85,B 0,C 180,E1 -5931.756,E2 -5931.756} C_VEL
LIN {X 0,Y 503.103,Z 338.391,A -85,B 0,C 180,E1 -5932.019,E2 -5932.019} C_VEL
LIN {X 0,Y 502.96,Z 346.989,A -85,B 0,C 180,E1 -5932.472,E2 -5932.472} C_VEL
LIN {X 0,Y 502.858,Z 355.5,A -85,B 0,C 180,E1 -5933.073,E2 -5933.073} C_VEL
LIN {X 0,Y 502.612,Z 362.983,A -85,B 0,C 180,E1 -5933.778,E2 -5933.778} C_VEL
LIN {X 0,Y 502.659,Z 369.636,A -85,B 0,C 180,E1 -5934.584,E2 -5934.584} C_VEL
LIN {X 0,Y 502.521,Z 374.732,A -85,B 0,C 180,E1 -5935.386,E2 -5935.386} C_VEL
LIN {X 0,Y 502.492,Z 379.651,A -85,B 0,C 180,E1 -5936.391,E2 -5936.391} C_VEL
LIN {X 0,Y 502.351,Z 382.53,A -85,B 0,C 180,E1 -5937.192,E2 -5937.192} C_VEL
LIN {X 0,Y 502.141,Z 385.371,A -85,B 0,C 180,E1 -5938.395,E2 -5938.395} C_VEL
LIN {X 0,Y 502.121,Z 386.403,A -85,B 0,C 180,E1 -5939.197,E2 -5939.197} C_VEL
LIN {X 0,Y 502.115,Z 386.757,A -85,B 0,C 180,E1 -5939.999,E2 -5939.999} C_VEL
LIN {X 0,Y 502.116,Z 386.441,A -85,B 0,C 180,E1 -5940.801,E2 -5940.801} C_VEL
LIN {X 0,Y 502.132,Z 385.449,A -85,B 0,C 180,E1 -5941.603,E2 -5941.603} C_VEL
LIN {X 0,Y 502.188,Z 383.749,A -85,B 0,C 180,E1 -5942.405,E2 -5942.405} C_VEL
LIN {X 0,Y 502.309,Z 381.299,A -85,B 0,C 180,E1 -5943.207,E2 -5943.207} C_VEL
LIN {X 0,Y 502.454,Z 378.021,A -85,B 0,C 180,E1 -5944.009,E2 -5944.009} C_VEL
LIN {X 0,Y 502.544,Z 372.642,A -85,B 0,C 180,E1 -5945.013,E2 -5945.013} C_VEL
LIN {X 0,Y 502.597,Z 366.884,A -85,B 0,C 180,E1 -5945.817,E2 -5945.817} C_VEL
LIN {X 0,Y 502.733,Z 359.842,A -85,B 0,C 180,E1 -5946.596,E2 -5946.596} C_VEL
LIN {X 0,Y 502.848,Z 352.378,A -85,B 0,C 180,E1 -5947.225,E2 -5947.225} C_VEL
LIN {X 0,Y 503.014,Z 344.707,A -85,B 0,C 180,E1 -5947.727,E2 -5947.727} C_VEL
LIN {X 0,Y 502.921,Z 335.234,A -85,B 0,C 180,E1 -5948.184,E2 -5948.184} C_VEL
LIN {X 0,Y 502.331,Z 331.17,A -85,B 0,C 180,E1 -5948.345,E2 -5948.345} C_VEL
LIN {X 0,Y 502.387,Z 323.299,A -85,B 0,C 180,E1 -5951.692,E2 -5951.692} C_VEL
LIN {X 0,Y 502.432,Z 315.203,A -85,B 0,C 180,E1 -5955.166,E2 -5955.166} C_VEL
LIN {X 0,Y 502.486,Z 308.616,A -85,B 0,C 180,E1 -5957.995,E2 -5957.995} C_VEL
LIN {X 0,Y 502.539,Z 301.838,A -85,B 0,C 180,E1 -5960.891,E2 -5960.891} C_VEL
LIN {X 0,Y 502.581,Z 294.776,A -85,B 0,C 180,E1 -5963.923,E2 -5963.923} C_VEL
LIN {X 0,Y 502.627,Z 287.361,A -85,B 0,C 180,E1 -5967.027,E2 -5967.027} C_VEL
LIN {X 0,Y 502.721,Z 281.868,A -85,B 0,C 180,E1 -5969.343,E2 -5969.343} C_VEL
LIN {X 0,Y 502.767,Z 281.854,A -85,B 0,C 180,E1 -5972.084,E2 -5972.084} C_VEL
LIN {X 0,Y 502.785,Z 281.857,A -85,B 0,C 180,E1 -5974.965,E2 -5974.965} C_VEL
LIN {X 0,Y 502.784,Z 281.855,A -85,B 0,C 180,E1 -5978.484,E2 -5978.484} C_VEL
LIN {X 0,Y 502.77,Z 281.859,A -85,B 0,C 180,E1 -5981.069,E2 -5981.069} C_VEL
LIN {X 0,Y 502.749,Z 281.858,A -85,B 0,C 180,E1 -5983.371,E2 -5983.371} C_VEL
LIN {X 0,Y 502.771,Z 281.855,A -85,B 0,C 180,E1 -5985.659,E2 -5985.659} C_VEL
LIN {X 0,Y 502.811,Z 281.851,A -85,B 0,C 180,E1 -5989.004,E2 -5989.004} C_VEL
LIN {X 0,Y 502.786,Z 281.857,A -85,B 0,C 180,E1 -5992.045,E2 -5992.045} C_VEL
LIN {X 0,Y 502.801,Z 281.852,A -85,B 0,C 180,E1 -5995.034,E2 -5995.034} C_VEL
LIN {X 0,Y 502.792,Z 281.853,A -85,B 0,C 180,E1 -5996.391,E2 -5996.391} C_VEL
LIN {X 0,Y 502.138,Z 281.935,A -85,B 0,C 180,E1 -5997.059,E2 -5997.059} C_VEL
LIN {X 0,Y 499.293,Z 282.293,A -85,B 0,C 180,E1 -5998.144,E2 -5998.144} C_VEL
LIN {X 0,Y 496.882,Z 282.596,A -85,B 0,C 180,E1 -5999.018,E2 -5999.018} C_VEL
LIN {X 0,Y 495.849,Z 282.723,A -85,B 0,C 180,E1 -5999.694,E2 -5999.694} C_VEL
LIN {X 0,Y 495.766,Z 282.732,A -85,B 0,C 180,E1 -5999.922,E2 -5999.922} C_VEL
LIN {X 0,Y 495.823,Z 282.725,A -85,B 0,C 180,E1 -6003.247,E2 -6003.247} C_VEL
LIN {X 0,Y 495.742,Z 282.735,A -85,B 0,C 180,E1 -6005.724,E2 -6005.724} C_VEL
LIN {X 0,Y 495.736,Z 282.732,A -85,B 0,C 180,E1 -6008.371,E2 -6008.371} C_VEL
LIN {X 0,Y 495.774,Z 282.732,A -85,B 0,C 180,E1 -6010.971,E2 -6010.971} C_VEL
LIN {X 0,Y 495.767,Z 282.729,A -85,B 0,C 180,E1 -6013.53,E2 -6013.53} C_VEL
LIN {X 0,Y 495.781,Z 282.726,A -85,B 0,C 180,E1 -6016.055,E2 -6016.055} C_VEL
LIN {X 0,Y 495.838,Z 282.725,A -85,B 0,C 180,E1 -6018.554,E2 -6018.554} C_VEL
LIN {X 0,Y 495.823,Z 282.721,A -85,B 0,C 180,E1 -6021.851,E2 -6021.851} C_VEL
LIN {X 0,Y 495.865,Z 282.721,A -85,B 0,C 180,E1 -6024.306,E2 -6024.306} C_VEL
LIN {X 0,Y 495.965,Z 282.703,A -85,B 0,C 180,E1 -6027.564,E2 -6027.564} C_VEL
LIN {X 0,Y 495.959,Z 282.71,A -85,B 0,C 180,E1 -6030,E2 -6030} C_VEL
LIN {X 0,Y 495.965,Z 282.703,A -85,B 0,C 180,E1 -6032.436,E2 -6032.436} C_VEL
LIN {X 0,Y 495.865,Z 282.722,A -85,B 0,C 180,E1 -6035.694,E2 -6035.694} C_VEL
LIN {X 0,Y 495.825,Z 282.722,A -85,B 0,C 180,E1 -6038.97,E2 -6038.97} C_VEL
LIN {X 0,Y 495.815,Z 282.722,A -85,B 0,C 180,E1 -6042.035,E2 -6042.035} C_VEL
LIN {X 0,Y 495.811,Z 282.726,A -85,B 0,C 180,E1 -6045.452,E2 -6045.452} C_VEL
LIN {X 0,Y 495.795,Z 282.725,A -85,B 0,C 180,E1 -6048.248,E2 -6048.248} C_VEL
LIN {X 0,Y 495.763,Z 282.732,A -85,B 0,C 180,E1 -6050.757,E2 -6050.757} C_VEL
LIN {X 0,Y 495.742,Z 282.732,A -85,B 0,C 180,E1 -6053.388,E2 -6053.388} C_VEL
LIN {X 0,Y 495.789,Z 282.728,A -85,B 0,C 180,E1 -6056.068,E2 -6056.068} C_VEL
LIN {X 0,Y 495.771,Z 282.73,A -85,B 0,C 180,E1 -6058.815,E2 -6058.815} C_VEL
LIN {X 0,Y 495.75,Z 282.733,A -85,B 0,C 180,E1 -6061.727,E2 -6061.727} C_VEL
LIN {X 0,Y 495.768,Z 282.728,A -85,B 0,C 180,E1 -6064.696,E2 -6064.696} C_VEL
LIN {X 0,Y 495.723,Z 282.738,A -85,B 0,C 180,E1 -6067.562,E2 -6067.562} C_VEL
LIN {X 0,Y 495.758,Z 282.729,A -85,B 0,C 180,E1 -6070.701,E2 -6070.701} C_VEL
LIN {X 0,Y 495.72,Z 282.735,A -85,B 0,C 180,E1 -6074.003,E2 -6074.003} C_VEL
LIN {X 0,Y 495.707,Z 282.74,A -85,B 0,C 180,E1 -6077.117,E2 -6077.117} C_VEL
LIN {X 0,Y 495.737,Z 282.731,A -85,B 0,C 180,E1 -6080.362,E2 -6080.362} C_VEL
LIN {X 0,Y 495.707,Z 282.735,A -85,B 0,C 180,E1 -6083.456,E2 -6083.456} C_VEL
LIN {X 0,Y 495.735,Z 282.734,A -85,B 0,C 180,E1 -6086.435,E2 -6086.435} C_VEL
LIN {X 0,Y 495.835,Z 282.813,A -85,B 0,C 180,E1 -6089.84,E2 -6089.84} C_VEL
LIN {X 0,Y 495.75,Z 287.533,A -85,B 0,C 180,E1 -6092.108,E2 -6092.108} C_VEL
LIN {X 0,Y 495.586,Z 293.994,A -85,B 0,C 180,E1 -6095.176,E2 -6095.176} C_VEL
LIN {X 0,Y 495.465,Z 300.825,A -85,B 0,C 180,E1 -6098.36,E2 -6098.36} C_VEL
LIN {X 0,Y 495.396,Z 306.426,A -85,B 0,C 180,E1 -6100.957,E2 -6100.957} C_VEL
LIN {X 0,Y 495.27,Z 312.011,A -85,B 0,C 180,E1 -6103.514,E2 -6103.514} C_VEL
LIN {X 0,Y 495.199,Z 317.583,A -85,B 0,C 180,E1 -6106.04,E2 -6106.04} C_VEL
LIN {X 0,Y 495.226,Z 323.134,A -85,B 0,C 180,E1 -6108.541,E2 -6108.541} C_VEL
LIN {X 0,Y 495.154,Z 329.58,A -85,B 0,C 180,E1 -6111.405,E2 -6111.405} C_VEL
LIN {X 0,Y 496.214,Z 338.686,A -85,B 0,C 180,E1 -6111.808,E2 -6111.808} C_VEL
LIN {X 0,Y 496.014,Z 348.418,A -85,B 0,C 180,E1 -6112.368,E2 -6112.368} C_VEL
LIN {X 0,Y 495.846,Z 357.667,A -85,B 0,C 180,E1 -6113.098,E2 -6113.098} C_VEL
LIN {X 0,Y 495.614,Z 365.351,A -85,B 0,C 180,E1 -6113.896,E2 -6113.896} C_VEL
LIN {X 0,Y 495.61,Z 371.442,A -85,B 0,C 180,E1 -6114.712,E2 -6114.712} C_VEL
LIN {X 0,Y 495.437,Z 377.319,A -85,B 0,C 180,E1 -6115.73,E2 -6115.73} C_VEL
LIN {X 0,Y 495.259,Z 381.649,A -85,B 0,C 180,E1 -6116.747,E2 -6116.747} C_VEL
LIN {X 0,Y 495.128,Z 384.191,A -85,B 0,C 180,E1 -6117.561,E2 -6117.561} C_VEL
LIN {X 0,Y 495.07,Z 385.983,A -85,B 0,C 180,E1 -6118.374,E2 -6118.374} C_VEL
LIN {X 0,Y 495.06,Z 387.078,A -85,B 0,C 180,E1 -6119.188,E2 -6119.188} C_VEL
LIN {X 0,Y 495.062,Z 387.506,A -85,B 0,C 180,E1 -6120.001,E2 -6120.001} C_VEL
LIN {X 0,Y 495.068,Z 387.271,A -85,B 0,C 180,E1 -6120.814,E2 -6120.814} C_VEL
LIN {X 0,Y 495.09,Z 386.37,A -85,B 0,C 180,E1 -6121.628,E2 -6121.628} C_VEL
LIN {X 0,Y 495.311,Z 383.7,A -85,B 0,C 180,E1 -6122.848,E2 -6122.848} C_VEL
LIN {X 0,Y 495.462,Z 380.978,A -85,B 0,C 180,E1 -6123.661,E2 -6123.661} C_VEL
LIN {X 0,Y 495.504,Z 376.405,A -85,B 0,C 180,E1 -6124.679,E2 -6124.679} C_VEL
LIN {X 0,Y 495.653,Z 371.583,A -85,B 0,C 180,E1 -6125.493,E2 -6125.493} C_VEL
LIN {X 0,Y 495.763,Z 365.494,A -85,B 0,C 180,E1 -6126.309,E2 -6126.309} C_VEL
LIN {X 0,Y 496.035,Z 358.615,A -85,B 0,C 180,E1 -6127.034,E2 -6127.034} C_VEL
LIN {X 0,Y 496.151,Z 350.663,A -85,B 0,C 180,E1 -6127.694,E2 -6127.694} C_VEL
LIN {X 0,Y 496.32,Z 341.928,A -85,B 0,C 180,E1 -6128.244,E2 -6128.244} C_VEL
LIN {X 0,Y 496.116,Z 335.676,A -85,B 0,C 180,E1 -6128.555,E2 -6128.555} C_VEL
LIN {X 0,Y 495.28,Z 330.817,A -85,B 0,C 180,E1 -6128.775,E2 -6128.775} C_VEL
LIN {X 0,Y 495.382,Z 324.254,A -85,B 0,C 180,E1 -6131.788,E2 -6131.788} C_VEL
LIN {X 0,Y 495.507,Z 316.69,A -85,B 0,C 180,E1 -6135.317,E2 -6135.317} C_VEL
LIN {X 0,Y 495.64,Z 310.686,A -85,B 0,C 180,E1 -6138.188,E2 -6138.188} C_VEL
LIN {X 0,Y 495.763,Z 305.339,A -85,B 0,C 180,E1 -6140.758,E2 -6140.758} C_VEL
LIN {X 0,Y 495.879,Z 299.9,A -85,B 0,C 180,E1 -6143.382,E2 -6143.382} C_VEL
LIN {X 0,Y 496.033,Z 294.456,A -85,B 0,C 180,E1 -6146.055,E2 -6146.055} C_VEL
LIN {X 0,Y 496.22,Z 288.996,A -85,B 0,C 180,E1 -6148.787,E2 -6148.787} C_VEL
LIN {X 0,Y 496.128,Z 285.396,A -85,B 0,C 180,E1 -6150.662,E2 -6150.662} C_VEL
LIN {X 0,Y 495.755,Z 282.735,A -85,B 0,C 180,E1 -6152.126,E2 -6152.126} C_VEL
LIN {X 0,Y 495.775,Z 282.733,A -85,B 0,C 180,E1 -6154.694,E2 -6154.694} C_VEL
LIN {X 0,Y 495.734,Z 282.737,A -85,B 0,C 180,E1 -6157.562,E2 -6157.562} C_VEL
LIN {X 0,Y 495.772,Z 282.732,A -85,B 0,C 180,E1 -6160.7,E2 -6160.7} C_VEL
LIN {X 0,Y 495.733,Z 282.737,A -85,B 0,C 180,E1 -6164.002,E2 -6164.002} C_VEL
LIN {X 0,Y 495.73,Z 282.737,A -85,B 0,C 180,E1 -6167.117,E2 -6167.117} C_VEL
LIN {X 0,Y 495.764,Z 282.733,A -85,B 0,C 180,E1 -6169.953,E2 -6169.953} C_VEL
LIN {X 0,Y 495.733,Z 282.738,A -85,B 0,C 180,E1 -6172.554,E2 -6172.554} C_VEL
LIN {X 0,Y 495.783,Z 282.732,A -85,B 0,C 180,E1 -6175.457,E2 -6175.457} C_VEL
LIN {X 0,Y 495.808,Z 282.848,A -85,B 0,C 180,E1 -6176.904,E2 -6176.904} C_VEL
LIN {X 0,Y 497.691,Z 291.051,A -85,B 0,C 180,E1 -6179.474,E2 -6179.474} C_VEL
LIN {X 0,Y 499.056,Z 298.144,A -85,B 0,C 180,E1 -6181.392,E2 -6181.392} C_VEL
LIN {X 0,Y 498.323,Z 307.885,A -85,B 0,C 180,E1 -6183.624,E2 -6183.624} C_VEL
LIN {X 0,Y 497.392,Z 321.476,A -85,B 0,C 180,E1 -6186.474,E2 -6186.474} C_VEL
LIN {X 0,Y 496.722,Z 336.679,A -85,B 0,C 180,E1 -6189.501,E2 -6189.501} C_VEL
LIN {X 0,Y 496.15,Z 353.517,A -85,B 0,C 180,E1 -6192.694,E2 -6192.694} C_VEL
LIN {X 0,Y 495.79,Z 370.008,A -85,B 0,C 180,E1 -6195.715,E2 -6195.715} C_VEL
LIN {X 0,Y 497.179,Z 383.134,A -85,B 0,C 180,E1 -6196.03,E2 -6196.03} C_VEL
LIN {X 0,Y 497.094,Z 395.775,A -85,B 0,C 180,E1 -6196.458,E2 -6196.458} C_VEL
LIN {X 0,Y 496.717,Z 408.025,A -85,B 0,C 180,E1 -6197.03,E2 -6197.03} C_VEL
LIN {X 0,Y 496.445,Z 419.459,A -85,B 0,C 180,E1 -6197.74,E2 -6197.74} C_VEL
LIN {X 0,Y 496.141,Z 430.01,A -85,B 0,C 180,E1 -6198.562,E2 -6198.562} C_VEL
LIN {X 0,Y 495.813,Z 440.644,A -85,B 0,C 180,E1 -6199.588,E2 -6199.588} C_VEL
LIN {X 0,Y 495.559,Z 449.219,A -85,B 0,C 180,E1 -6200.614,E2 -6200.614} C_VEL
LIN {X 0,Y 495.359,Z 457.591,A -85,B 0,C 180,E1 -6201.843,E2 -6201.843} C_VEL
LIN {X 0,Y 495.253,Z 464.322,A -85,B 0,C 180,E1 -6203.072,E2 -6203.072} C_VEL
LIN {X 0,Y 495.186,Z 469.662,A -85,B 0,C 180,E1 -6204.298,E2 -6204.298} C_VEL
LIN {X 0,Y 495.1,Z 473.792,A -85,B 0,C 180,E1 -6205.522,E2 -6205.522} C_VEL
LIN {X 0,Y 495.155,Z 476.85,A -85,B 0,C 180,E1 -6206.745,E2 -6206.745} C_VEL
LIN {X 0,Y 495.061,Z 478.301,A -85,B 0,C 180,E1 -6207.559,E2 -6207.559} C_VEL
LIN {X 0,Y 494.969,Z 479.971,A -85,B 0,C 180,E1 -6209.186,E2 -6209.186} C_VEL
LIN {X 0,Y 494.969,Z 480.207,A -85,B 0,C 180,E1 -6210,E2 -6210} C_VEL
LIN {X 0,Y 494.967,Z 479.993,A -85,B 0,C 180,E1 -6210.814,E2 -6210.814} C_VEL
LIN {X 0,Y 495.061,Z 478.378,A -85,B 0,C 180,E1 -6212.441,E2 -6212.441} C_VEL
LIN {X 0,Y 495.138,Z 476.947,A -85,B 0,C 180,E1 -6213.255,E2 -6213.255} C_VEL
LIN {X 0,Y 495.08,Z 473.937,A -85,B 0,C 180,E1 -6214.478,E2 -6214.478} C_VEL
LIN {X 0,Y 495.177,Z 468.723,A -85,B 0,C 180,E1 -6215.985,E2 -6215.985} C_VEL
LIN {X 0,Y 495.271,Z 462.529,A -85,B 0,C 180,E1 -6217.337,E2 -6217.337} C_VEL
LIN {X 0,Y 495.451,Z 455.372,A -85,B 0,C 180,E1 -6218.566,E2 -6218.566} C_VEL
LIN {X 0,Y 495.628,Z 446.407,A -85,B 0,C 180,E1 -6219.797,E2 -6219.797} C_VEL
LIN {X 0,Y 495.96,Z 437.216,A -85,B 0,C 180,E1 -6220.822,E2 -6220.822} C_VEL
LIN {X 0,Y 496.301,Z 426.99,A -85,B 0,C 180,E1 -6221.745,E2 -6221.745} C_VEL
LIN {X 0,Y 496.569,Z 416.082,A -85,B 0,C 180,E1 -6222.537,E2 -6222.537} C_VEL
LIN {X 0,Y 496.931,Z 403.816,A -85,B 0,C 180,E1 -6223.235,E2 -6223.235} C_VEL
LIN {X 0,Y 497.232,Z 391.597,A -85,B 0,C 180,E1 -6223.747,E2 -6223.747} C_VEL
LIN {X 0,Y 497.224,Z 382.876,A -85,B 0,C 180,E1 -6224.021,E2 -6224.021} C_VEL
LIN {X 0,Y 495.823,Z 370.314,A -85,B 0,C 180,E1 -6224.336,E2 -6224.336} C_VEL
LIN {X 0,Y 496.265,Z 353.232,A -85,B 0,C 180,E1 -6227.514,E2 -6227.514} C_VEL
LIN {X 0,Y 496.917,Z 334.742,A -85,B 0,C 180,E1 -6231.019,E2 -6231.019} C_VEL
LIN {X 0,Y 497.631,Z 318.524,A -85,B 0,C 180,E1 -6234.178,E2 -6234.178} C_VEL
LIN {X 0,Y 498.487,Z 302.667,A -85,B 0,C 180,E1 -6237.349,E2 -6237.349} C_VEL
LIN {X 0,Y 498.661,Z 296.43,A -85,B 0,C 180,E1 -6238.632,E2 -6238.632} C_VEL
LIN {X 0,Y 496.361,Z 285.445,A -85,B 0,C 180,E1 -6241.118,E2 -6241.118} C_VEL
LIN {X 0,Y 495.747,Z 282.735,A -85,B 0,C 180,E1 -6241.767,E2 -6241.767} C_VEL
LIN {X 0,Y 495.767,Z 282.733,A -85,B 0,C 180,E1 -6244.693,E2 -6244.693} C_VEL
LIN {X 0,Y 495.734,Z 282.738,A -85,B 0,C 180,E1 -6247.561,E2 -6247.561} C_VEL
LIN {X 0,Y 495.771,Z 282.732,A -85,B 0,C 180,E1 -6250.7,E2 -6250.7} C_VEL
LIN {X 0,Y 495.739,Z 282.736,A -85,B 0,C 180,E1 -6254.001,E2 -6254.001} C_VEL
LIN {X 0,Y 495.731,Z 282.738,A -85,B 0,C 180,E1 -6257.117,E2 -6257.117} C_VEL
LIN {X 0,Y 495.764,Z 282.732,A -85,B 0,C 180,E1 -6259.953,E2 -6259.953} C_VEL
LIN {X 0,Y 495.733,Z 282.737,A -85,B 0,C 180,E1 -6262.553,E2 -6262.553} C_VEL
LIN {X 0,Y 495.776,Z 282.734,A -85,B 0,C 180,E1 -6265.456,E2 -6265.456} C_VEL
LIN {X 0,Y 495.76,Z 282.736,A -85,B 0,C 180,E1 -6268.363,E2 -6268.363} C_VEL
LIN {X 0,Y 495.624,Z 282.753,A -85,B 0,C 180,E1 -6271.175,E2 -6271.175} C_VEL
LIN {X 0,Y 495.526,Z 282.874,A -85,B 0,C 180,E1 -6271.837,E2 -6271.837} C_VEL
LIN {X 0,Y 495.477,Z 291.237,A -85,B 0,C 180,E1 -6274.815,E2 -6274.815} C_VEL
LIN {X 0,Y 495.508,Z 298.312,A -85,B 0,C 180,E1 -6277.482,E2 -6277.482} C_VEL
LIN {X 0,Y 495.473,Z 305.999,A -85,B 0,C 180,E1 -6280.528,E2 -6280.528} C_VEL
LIN {X 0,Y 495.429,Z 312.25,A -85,B 0,C 180,E1 -6283.093,E2 -6283.093} C_VEL
LIN {X 0,Y 495.422,Z 318.42,A -85,B 0,C 180,E1 -6285.625,E2 -6285.625} C_VEL
LIN {X 0,Y 495.448,Z 325.33,A -85,B 0,C 180,E1 -6288.544,E2 -6288.544} C_VEL
LIN {X 0,Y 495.396,Z 332.614,A -85,B 0,C 180,E1 -6291.638,E2 -6291.638} C_VEL
LIN {X 0,Y 496.101,Z 339.053,A -85,B 0,C 180,E1 -6291.906,E2 -6291.906} C_VEL
LIN {X 0,Y 495.969,Z 347.636,A -85,B 0,C 180,E1 -6292.365,E2 -6292.365} C_VEL
LIN {X 0,Y 495.881,Z 355.033,A -85,B 0,C 180,E1 -6292.884,E2 -6292.884} C_VEL
LIN {X 0,Y 495.669,Z 361.719,A -85,B 0,C 180,E1 -6293.486,E2 -6293.486} C_VEL
LIN {X 0,Y 495.608,Z 368.753,A -85,B 0,C 180,E1 -6294.302,E2 -6294.302} C_VEL
LIN {X 0,Y 495.48,Z 374.269,A -85,B 0,C 180,E1 -6295.117,E2 -6295.117} C_VEL
LIN {X 0,Y 495.421,Z 378.506,A -85,B 0,C 180,E1 -6295.932,E2 -6295.932} C_VEL
LIN {X 0,Y 495.283,Z 381.816,A -85,B 0,C 180,E1 -6296.745,E2 -6296.745} C_VEL
LIN {X 0,Y 495.141,Z 384.301,A -85,B 0,C 180,E1 -6297.558,E2 -6297.558} C_VEL
LIN {X 0,Y 495.075,Z 386.033,A -85,B 0,C 180,E1 -6298.372,E2 -6298.372} C_VEL
LIN {X 0,Y 495.054,Z 387.064,A -85,B 0,C 180,E1 -6299.186,E2 -6299.186} C_VEL
LIN {X 0,Y 495.047,Z 387.415,A -85,B 0,C 180,E1 -6299.999,E2 -6299.999} C_VEL
LIN {X 0,Y 495.047,Z 387.093,A -85,B 0,C 180,E1 -6300.812,E2 -6300.812} C_VEL
LIN {X 0,Y 495.064,Z 386.093,A -85,B 0,C 180,E1 -6301.626,E2 -6301.626} C_VEL
LIN {X 0,Y 495.125,Z 384.383,A -85,B 0,C 180,E1 -6302.439,E2 -6302.439} C_VEL
LIN {X 0,Y 495.257,Z 381.913,A -85,B 0,C 180,E1 -6303.253,E2 -6303.253} C_VEL
LIN {X 0,Y 495.419,Z 378.621,A -85,B 0,C 180,E1 -6304.066,E2 -6304.066} C_VEL
LIN {X 0,Y 495.512,Z 373.223,A -85,B 0,C 180,E1 -6305.085,E2 -6305.085} C_VEL
LIN {X 0,Y 495.569,Z 367.439,A -85,B 0,C 180,E1 -6305.9,E2 -6305.9} C_VEL
LIN {X 0,Y 495.71,Z 360.376,A -85,B 0,C 180,E1 -6306.69,E2 -6306.69} C_VEL
LIN {X 0,Y 495.835,Z 352.878,A -85,B 0,C 180,E1 -6307.328,E2 -6307.328} C_VEL
LIN {X 0,Y 495.997,Z 345.187,A -85,B 0,C 180,E1 -6307.837,E2 -6307.837} C_VEL
LIN {X 0,Y 495.874,Z 335.657,A -85,B 0,C 180,E1 -6308.301,E2 -6308.301} C_VEL
LIN {X 0,Y 495.306,Z 331.703,A -85,B 0,C 180,E1 -6308.464,E2 -6308.464} C_VEL
LIN {X 0,Y 495.347,Z 323.949,A -85,B 0,C 180,E1 -6311.769,E2 -6311.769} C_VEL
LIN {X 0,Y 495.407,Z 315.782,A -85,B 0,C 180,E1 -6315.275,E2 -6315.275} C_VEL
LIN {X 0,Y 495.447,Z 307.993,A -85,B 0,C 180,E1 -6318.611,E2 -6318.611} C_VEL
LIN {X 0,Y 495.476,Z 301.94,A -85,B 0,C 180,E1 -6321.203,E2 -6321.203} C_VEL
LIN {X 0,Y 495.517,Z 294.706,A -85,B 0,C 180,E1 -6324.286,E2 -6324.286} C_VEL
LIN {X 0,Y 495.594,Z 287.199,A -85,B 0,C 180,E1 -6327.442,E2 -6327.442} C_VEL
LIN {X 0,Y 495.684,Z 282.745,A -85,B 0,C 180,E1 -6329.342,E2 -6329.342} C_VEL
LIN {X 0,Y 495.743,Z 282.73,A -85,B 0,C 180,E1 -6332.595,E2 -6332.595} C_VEL
LIN {X 0,Y 495.736,Z 282.733,A -85,B 0,C 180,E1 -6335.537,E2 -6335.537} C_VEL
LIN {X 0,Y 495.751,Z 282.733,A -85,B 0,C 180,E1 -6338.766,E2 -6338.766} C_VEL
LIN {X 0,Y 495.737,Z 282.731,A -85,B 0,C 180,E1 -6341.781,E2 -6341.781} C_VEL
LIN {X 0,Y 495.729,Z 282.734,A -85,B 0,C 180,E1 -6345.14,E2 -6345.14} C_VEL
LIN {X 0,Y 495.748,Z 282.734,A -85,B 0,C 180,E1 -6348.218,E2 -6348.218} C_VEL
LIN {X 0,Y 495.743,Z 282.731,A -85,B 0,C 180,E1 -6351.407,E2 -6351.407} C_VEL
LIN {X 0,Y 495.749,Z 282.733,A -85,B 0,C 180,E1 -6354.462,E2 -6354.462} C_VEL
LIN {X 0,Y 495.76,Z 282.731,A -85,B 0,C 180,E1 -6357.405,E2 -6357.405} C_VEL
LIN {X 0,Y 495.766,Z 282.732,A -85,B 0,C 180,E1 -6359.922,E2 -6359.922} C_VEL
LIN {X 0,Y 495.109,Z 282.811,A -85,B 0,C 180,E1 -6360.6,E2 -6360.6} C_VEL
LIN {X 0,Y 492.281,Z 283.166,A -85,B 0,C 180,E1 -6361.7,E2 -6361.7} C_VEL
LIN {X 0,Y 489.883,Z 283.463,A -85,B 0,C 180,E1 -6362.587,E2 -6362.587} C_VEL
LIN {X 0,Y 488.845,Z 283.595,A -85,B 0,C 180,E1 -6363.272,E2 -6363.272} C_VEL
LIN {X 0,Y 488.757,Z 283.605,A -85,B 0,C 180,E1 -6363.504,E2 -6363.504} C_VEL
LIN {X 0,Y 488.683,Z 283.611,A -85,B 0,C 180,E1 -6366.254,E2 -6366.254} C_VEL
LIN {X 0,Y 488.735,Z 283.608,A -85,B 0,C 180,E1 -6369.175,E2 -6369.175} C_VEL
LIN {X 0,Y 488.748,Z 283.604,A -85,B 0,C 180,E1 -6371.627,E2 -6371.627} C_VEL
LIN {X 0,Y 488.75,Z 283.605,A -85,B 0,C 180,E1 -6374.999,E2 -6374.999} C_VEL
LIN {X 0,Y 488.792,Z 283.601,A -85,B 0,C 180,E1 -6378.387,E2 -6378.387} C_VEL
LIN {X 0,Y 488.772,Z 283.599,A -85,B 0,C 180,E1 -6381.733,E2 -6381.733} C_VEL
LIN {X 0,Y 488.822,Z 283.599,A -85,B 0,C 180,E1 -6384.224,E2 -6384.224} C_VEL
LIN {X 0,Y 488.931,Z 283.579,A -85,B 0,C 180,E1 -6387.528,E2 -6387.528} C_VEL
LIN {X 0,Y 488.928,Z 283.586,A -85,B 0,C 180,E1 -6390,E2 -6390} C_VEL
LIN {X 0,Y 488.931,Z 283.579,A -85,B 0,C 180,E1 -6392.472,E2 -6392.472} C_VEL
LIN {X 0,Y 488.822,Z 283.598,A -85,B 0,C 180,E1 -6395.776,E2 -6395.776} C_VEL
LIN {X 0,Y 488.772,Z 283.599,A -85,B 0,C 180,E1 -6398.267,E2 -6398.267} C_VEL
LIN {X 0,Y 488.793,Z 283.6,A -85,B 0,C 180,E1 -6401.613,E2 -6401.613} C_VEL
LIN {X 0,Y 488.75,Z 283.605,A -85,B 0,C 180,E1 -6405.001,E2 -6405.001} C_VEL
LIN {X 0,Y 488.743,Z 283.605,A -85,B 0,C 180,E1 -6408.443,E2 -6408.443} C_VEL
LIN {X 0,Y 488.697,Z 283.613,A -85,B 0,C 180,E1 -6411.071,E2 -6411.071} C_VEL
LIN {X 0,Y 488.683,Z 283.611,A -85,B 0,C 180,E1 -6413.746,E2 -6413.746} C_VEL
LIN {X 0,Y 488.789,Z 283.599,A -85,B 0,C 180,E1 -6416.946,E2 -6416.946} C_VEL
LIN {X 0,Y 488.709,Z 283.611,A -85,B 0,C 180,E1 -6420.366,E2 -6420.366} C_VEL
LIN {X 0,Y 488.727,Z 283.607,A -85,B 0,C 180,E1 -6423.486,E2 -6423.486} C_VEL
LIN {X 0,Y 488.68,Z 283.613,A -85,B 0,C 180,E1 -6426.357,E2 -6426.357} C_VEL
LIN {X 0,Y 488.693,Z 283.611,A -85,B 0,C 180,E1 -6429.255,E2 -6429.255} C_VEL
LIN {X 0,Y 488.699,Z 283.613,A -85,B 0,C 180,E1 -6431.601,E2 -6431.601} C_VEL
LIN {X 0,Y 488.693,Z 283.61,A -85,B 0,C 180,E1 -6434.804,E2 -6434.804} C_VEL
LIN {X 0,Y 488.68,Z 283.613,A -85,B 0,C 180,E1 -6437.475,E2 -6437.475} C_VEL
LIN {X 0,Y 488.687,Z 283.612,A -85,B 0,C 180,E1 -6440.746,E2 -6440.746} C_VEL
LIN {X 0,Y 488.659,Z 283.612,A -85,B 0,C 180,E1 -6443.868,E2 -6443.868} C_VEL
LIN {X 0,Y 488.696,Z 283.613,A -85,B 0,C 180,E1 -6446.876,E2 -6446.876} C_VEL
LIN {X 0,Y 488.792,Z 283.673,A -85,B 0,C 180,E1 -6449.787,E2 -6449.787} C_VEL
LIN {X 0,Y 488.686,Z 289.464,A -85,B 0,C 180,E1 -6452.601,E2 -6452.601} C_VEL
LIN {X 0,Y 488.526,Z 295.243,A -85,B 0,C 180,E1 -6455.344,E2 -6455.344} C_VEL
LIN {X 0,Y 488.44,Z 300.936,A -85,B 0,C 180,E1 -6458.032,E2 -6458.032} C_VEL
LIN {X 0,Y 488.349,Z 306.578,A -85,B 0,C 180,E1 -6460.672,E2 -6460.672} C_VEL
LIN {X 0,Y 488.231,Z 312.211,A -85,B 0,C 180,E1 -6463.269,E2 -6463.269} C_VEL
LIN {X 0,Y 488.146,Z 317.808,A -85,B 0,C 180,E1 -6465.834,E2 -6465.834} C_VEL
LIN {X 0,Y 488.179,Z 323.4,A -85,B 0,C 180,E1 -6468.374,E2 -6468.374} C_VEL
LIN {X 0,Y 488.077,Z 329.838,A -85,B 0,C 180,E1 -6471.253,E2 -6471.253} C_VEL
LIN {X 0,Y 489.246,Z 339.433,A -85,B 0,C 180,E1 -6471.69,E2 -6471.69} C_VEL
LIN {X 0,Y 489.018,Z 349.059,A -85,B 0,C 180,E1 -6472.258,E2 -6472.258} C_VEL
LIN {X 0,Y 488.856,Z 356.873,A -85,B 0,C 180,E1 -6472.874,E2 -6472.874} C_VEL
LIN {X 0,Y 488.567,Z 364.146,A -85,B 0,C 180,E1 -6473.6,E2 -6473.6} C_VEL
LIN {X 0,Y 488.552,Z 370.64,A -85,B 0,C 180,E1 -6474.429,E2 -6474.429} C_VEL
LIN {X 0,Y 488.437,Z 376.867,A -85,B 0,C 180,E1 -6475.462,E2 -6475.462} C_VEL
LIN {X 0,Y 488.273,Z 380.683,A -85,B 0,C 180,E1 -6476.287,E2 -6476.287} C_VEL
LIN {X 0,Y 488.257,Z 383.627,A -85,B 0,C 180,E1 -6477.113,E2 -6477.113} C_VEL
LIN {X 0,Y 488.068,Z 384.822,A -85,B 0,C 180,E1 -6477.525,E2 -6477.525} C_VEL
LIN {X 0,Y 488.004,Z 386.631,A -85,B 0,C 180,E1 -6478.351,E2 -6478.351} C_VEL
LIN {X 0,Y 487.993,Z 387.741,A -85,B 0,C 180,E1 -6479.176,E2 -6479.176} C_VEL
LIN {X 0,Y 487.995,Z 388.182,A -85,B 0,C 180,E1 -6480.001,E2 -6480.001} C_VEL
LIN {X 0,Y 488.003,Z 387.959,A -85,B 0,C 180,E1 -6480.826,E2 -6480.826} C_VEL
LIN {X 0,Y 488.029,Z 387.069,A -85,B 0,C 180,E1 -6481.651,E2 -6481.651} C_VEL
LIN {X 0,Y 488.268,Z 384.415,A -85,B 0,C 180,E1 -6482.889,E2 -6482.889} C_VEL
LIN {X 0,Y 488.431,Z 381.704,A -85,B 0,C 180,E1 -6483.714,E2 -6483.714} C_VEL
LIN {X 0,Y 488.479,Z 377.152,A -85,B 0,C 180,E1 -6484.746,E2 -6484.746} C_VEL
LIN {X 0,Y 488.628,Z 370.978,A -85,B 0,C 180,E1 -6485.779,E2 -6485.779} C_VEL
LIN {X 0,Y 488.815,Z 363.354,A -85,B 0,C 180,E1 -6486.739,E2 -6486.739} C_VEL
LIN {X 0,Y 489.135,Z 355.24,A -85,B 0,C 180,E1 -6487.515,E2 -6487.515} C_VEL
LIN {X 0,Y 489.296,Z 346.68,A -85,B 0,C 180,E1 -6488.145,E2 -6488.145} C_VEL
LIN {X 0,Y 489.397,Z 338.125,A -85,B 0,C 180,E1 -6488.621,E2 -6488.621} C_VEL
LIN {X 0,Y 488.223,Z 331.244,A -85,B 0,C 180,E1 -6488.955,E2 -6488.955} C_VEL
LIN {X 0,Y 488.344,Z 324.985,A -85,B 0,C 180,E1 -6491.868,E2 -6491.868} C_VEL
LIN {X 0,Y 488.49,Z 317.431,A -85,B 0,C 180,E1 -6495.432,E2 -6495.432} C_VEL
LIN {X 0,Y 488.624,Z 311.152,A -85,B 0,C 180,E1 -6498.448,E2 -6498.448} C_VEL
LIN {X 0,Y 488.749,Z 305.791,A -85,B 0,C 180,E1 -6501.07,E2 -6501.07} C_VEL
LIN {X 0,Y 488.894,Z 300.387,A -85,B 0,C 180,E1 -6503.736,E2 -6503.736} C_VEL
LIN {X 0,Y 489.089,Z 294.98,A -85,B 0,C 180,E1 -6506.453,E2 -6506.453} C_VEL
LIN {X 0,Y 489.263,Z 289.595,A -85,B 0,C 180,E1 -6509.236,E2 -6509.236} C_VEL
LIN {X 0,Y 489.098,Z 286.014,A -85,B 0,C 180,E1 -6511.152,E2 -6511.152} C_VEL
LIN {X 0,Y 488.727,Z 283.611,A -85,B 0,C 180,E1 -6512.512,E2 -6512.512} C_VEL
LIN {X 0,Y 488.723,Z 283.611,A -85,B 0,C 180,E1 -6515.115,E2 -6515.115} C_VEL
LIN {X 0,Y 488.685,Z 283.616,A -85,B 0,C 180,E1 -6518.2,E2 -6518.2} C_VEL
LIN {X 0,Y 488.724,Z 283.61,A -85,B 0,C 180,E1 -6520.345,E2 -6520.345} C_VEL
LIN {X 0,Y 488.689,Z 283.614,A -85,B 0,C 180,E1 -6523.655,E2 -6523.655} C_VEL
LIN {X 0,Y 488.689,Z 283.616,A -85,B 0,C 180,E1 -6526.346,E2 -6526.346} C_VEL
LIN {X 0,Y 488.738,Z 283.609,A -85,B 0,C 180,E1 -6529.677,E2 -6529.677} C_VEL
LIN {X 0,Y 488.684,Z 283.616,A -85,B 0,C 180,E1 -6532.841,E2 -6532.841} C_VEL
LIN {X 0,Y 488.735,Z 283.611,A -85,B 0,C 180,E1 -6535.887,E2 -6535.887} C_VEL
LIN {X 0,Y 488.76,Z 283.759,A -85,B 0,C 180,E1 -6536.329,E2 -6536.329} C_VEL
LIN {X 0,Y 490.213,Z 289.961,A -85,B 0,C 180,E1 -6538.447,E2 -6538.447} C_VEL
LIN {X 0,Y 491.851,Z 297.465,A -85,B 0,C 180,E1 -6540.649,E2 -6540.649} C_VEL
LIN {X 0,Y 492.214,Z 300.386,A -85,B 0,C 180,E1 -6541.424,E2 -6541.424} C_VEL
LIN {X 0,Y 491.386,Z 310.099,A -85,B 0,C 180,E1 -6543.681,E2 -6543.681} C_VEL
LIN {X 0,Y 490.264,Z 324.957,A -85,B 0,C 180,E1 -6546.876,E2 -6546.876} C_VEL
LIN {X 0,Y 489.672,Z 338.598,A -85,B 0,C 180,E1 -6549.632,E2 -6549.632} C_VEL
LIN {X 0,Y 489.045,Z 355.358,A -85,B 0,C 180,E1 -6552.866,E2 -6552.866} C_VEL
LIN {X 0,Y 488.749,Z 369.628,A -85,B 0,C 180,E1 -6555.532,E2 -6555.532} C_VEL
LIN {X 0,Y 490.301,Z 385.406,A -85,B 0,C 180,E1 -6555.949,E2 -6555.949} C_VEL
LIN {X 0,Y 490.054,Z 398.062,A -85,B 0,C 180,E1 -6556.418,E2 -6556.418} C_VEL
LIN {X 0,Y 489.633,Z 410.772,A -85,B 0,C 180,E1 -6557.071,E2 -6557.071} C_VEL
LIN {X 0,Y 489.384,Z 422.434,A -85,B 0,C 180,E1 -6557.857,E2 -6557.857} C_VEL
LIN {X 0,Y 488.961,Z 433.579,A -85,B 0,C 180,E1 -6558.811,E2 -6558.811} C_VEL
LIN {X 0,Y 488.625,Z 443.394,A -85,B 0,C 180,E1 -6559.852,E2 -6559.852} C_VEL
LIN {X 0,Y 488.411,Z 451.418,A -85,B 0,C 180,E1 -6560.893,E2 -6560.893} C_VEL
LIN {X 0,Y 488.234,Z 459.22,A -85,B 0,C 180,E1 -6562.14,E2 -6562.14} C_VEL
LIN {X 0,Y 488.102,Z 465.856,A -85,B 0,C 180,E1 -6563.47,E2 -6563.47} C_VEL
LIN {X 0,Y 488.063,Z 470.423,A -85,B 0,C 180,E1 -6564.629,E2 -6564.629} C_VEL
LIN {X 0,Y 488.093,Z 474.215,A -85,B 0,C 180,E1 -6565.871,E2 -6565.871} C_VEL
LIN {X 0,Y 488.074,Z 476.168,A -85,B 0,C 180,E1 -6566.698,E2 -6566.698} C_VEL
LIN {X 0,Y 488,Z 477.633,A -85,B 0,C 180,E1 -6567.524,E2 -6567.524} C_VEL
LIN {X 0,Y 487.899,Z 479.314,A -85,B 0,C 180,E1 -6569.175,E2 -6569.175} C_VEL
LIN {X 0,Y 487.899,Z 479.555,A -85,B 0,C 180,E1 -6570,E2 -6570} C_VEL
LIN {X 0,Y 487.896,Z 479.342,A -85,B 0,C 180,E1 -6570.825,E2 -6570.825} C_VEL
LIN {X 0,Y 488,Z 477.729,A -85,B 0,C 180,E1 -6572.476,E2 -6572.476} C_VEL
LIN {X 0,Y 488.058,Z 476.29,A -85,B 0,C 180,E1 -6573.302,E2 -6573.302} C_VEL
LIN {X 0,Y 487.985,Z 473.27,A -85,B 0,C 180,E1 -6574.543,E2 -6574.543} C_VEL
LIN {X 0,Y 488.099,Z 469.181,A -85,B 0,C 180,E1 -6575.785,E2 -6575.785} C_VEL
LIN {X 0,Y 488.181,Z 462.852,A -85,B 0,C 180,E1 -6577.237,E2 -6577.237} C_VEL
LIN {X 0,Y 488.353,Z 455.948,A -85,B 0,C 180,E1 -6578.483,E2 -6578.483} C_VEL
LIN {X 0,Y 488.481,Z 448.871,A -85,B 0,C 180,E1 -6579.524,E2 -6579.524} C_VEL
LIN {X 0,Y 488.775,Z 440.332,A -85,B 0,C 180,E1 -6580.564,E2 -6580.564} C_VEL
LIN {X 0,Y 489.122,Z 429.74,A -85,B 0,C 180,E1 -6581.605,E2 -6581.605} C_VEL
LIN {X 0,Y 489.431,Z 418.968,A -85,B 0,C 180,E1 -6582.458,E2 -6582.458} C_VEL
LIN {X 0,Y 489.843,Z 406.756,A -85,B 0,C 180,E1 -6583.213,E2 -6583.213} C_VEL
LIN {X 0,Y 490.177,Z 394.321,A -85,B 0,C 180,E1 -6583.79,E2 -6583.79} C_VEL
LIN {X 0,Y 490.232,Z 383.451,A -85,B 0,C 180,E1 -6584.159,E2 -6584.159} C_VEL
LIN {X 0,Y 488.803,Z 370.133,A -85,B 0,C 180,E1 -6584.493,E2 -6584.493} C_VEL
LIN {X 0,Y 489.312,Z 351.735,A -85,B 0,C 180,E1 -6587.987,E2 -6587.987} C_VEL
LIN {X 0,Y 489.994,Z 333.724,A -85,B 0,C 180,E1 -6591.48,E2 -6591.48} C_VEL
LIN {X 0,Y 490.803,Z 317.229,A -85,B 0,C 180,E1 -6594.762,E2 -6594.762} C_VEL
LIN {X 0,Y 491.791,Z 300.708,A -85,B 0,C 180,E1 -6598.138,E2 -6598.138} C_VEL
LIN {X 0,Y 491.502,Z 296.311,A -85,B 0,C 180,E1 -6599.089,E2 -6599.089} C_VEL
LIN {X 0,Y 489.046,Z 285.356,A -85,B 0,C 180,E1 -6601.637,E2 -6601.637} C_VEL
LIN {X 0,Y 488.706,Z 283.613,A -85,B 0,C 180,E1 -6602.08,E2 -6602.08} C_VEL
LIN {X 0,Y 488.719,Z 283.611,A -85,B 0,C 180,E1 -6605.115,E2 -6605.115} C_VEL
LIN {X 0,Y 488.685,Z 283.615,A -85,B 0,C 180,E1 -6608.2,E2 -6608.2} C_VEL
LIN {X 0,Y 488.724,Z 283.61,A -85,B 0,C 180,E1 -6610.344,E2 -6610.344} C_VEL
LIN {X 0,Y 488.692,Z 283.613,A -85,B 0,C 180,E1 -6613.654,E2 -6613.654} C_VEL
LIN {X 0,Y 488.692,Z 283.612,A -85,B 0,C 180,E1 -6616.345,E2 -6616.345} C_VEL
LIN {X 0,Y 488.739,Z 283.606,A -85,B 0,C 180,E1 -6619.676,E2 -6619.676} C_VEL
LIN {X 0,Y 488.685,Z 283.614,A -85,B 0,C 180,E1 -6622.841,E2 -6622.841} C_VEL
LIN {X 0,Y 488.729,Z 283.61,A -85,B 0,C 180,E1 -6625.886,E2 -6625.886} C_VEL
LIN {X 0,Y 488.686,Z 283.618,A -85,B 0,C 180,E1 -6628.819,E2 -6628.819} C_VEL
LIN {X 0,Y 488.505,Z 283.642,A -85,B 0,C 180,E1 -6631.714,E2 -6631.714} C_VEL
LIN {X 0,Y 488.456,Z 292.82,A -85,B 0,C 180,E1 -6635.021,E2 -6635.021} C_VEL
LIN {X 0,Y 488.464,Z 300.735,A -85,B 0,C 180,E1 -6638.031,E2 -6638.031} C_VEL
LIN {X 0,Y 488.432,Z 308.305,A -85,B 0,C 180,E1 -6641.109,E2 -6641.109} C_VEL
LIN {X 0,Y 488.42,Z 315.803,A -85,B 0,C 180,E1 -6644.133,E2 -6644.133} C_VEL
LIN {X 0,Y 488.354,Z 322.909,A -85,B 0,C 180,E1 -6647.11,E2 -6647.11} C_VEL
LIN {X 0,Y 488.359,Z 327.879,A -85,B 0,C 180,E1 -6649.216,E2 -6649.216} C_VEL
LIN {X 0,Y 488.368,Z 333.287,A -85,B 0,C 180,E1 -6651.517,E2 -6651.517} C_VEL
LIN {X 0,Y 489.102,Z 339.754,A -85,B 0,C 180,E1 -6651.789,E2 -6651.789} C_VEL
LIN {X 0,Y 488.965,Z 348.323,A -85,B 0,C 180,E1 -6652.255,E2 -6652.255} C_VEL
LIN {X 0,Y 488.882,Z 356.011,A -85,B 0,C 180,E1 -6652.805,E2 -6652.805} C_VEL
LIN {X 0,Y 488.563,Z 364.319,A -85,B 0,C 180,E1 -6653.598,E2 -6653.598} C_VEL
LIN {X 0,Y 488.625,Z 370.974,A -85,B 0,C 180,E1 -6654.428,E2 -6654.428} C_VEL
LIN {X 0,Y 488.457,Z 376.076,A -85,B 0,C 180,E1 -6655.253,E2 -6655.253} C_VEL
LIN {X 0,Y 488.43,Z 380.994,A -85,B 0,C 180,E1 -6656.286,E2 -6656.286} C_VEL
LIN {X 0,Y 488.264,Z 383.875,A -85,B 0,C 180,E1 -6657.111,E2 -6657.111} C_VEL
LIN {X 0,Y 488.012,Z 386.713,A -85,B 0,C 180,E1 -6658.348,E2 -6658.348} C_VEL
LIN {X 0,Y 487.987,Z 387.736,A -85,B 0,C 180,E1 -6659.174,E2 -6659.174} C_VEL
LIN {X 0,Y 487.978,Z 388.078,A -85,B 0,C 180,E1 -6659.999,E2 -6659.999} C_VEL
LIN {X 0,Y 487.979,Z 387.745,A -85,B 0,C 180,E1 -6660.824,E2 -6660.824} C_VEL
LIN {X 0,Y 487.997,Z 386.731,A -85,B 0,C 180,E1 -6661.649,E2 -6661.649} C_VEL
LIN {X 0,Y 488.065,Z 385.003,A -85,B 0,C 180,E1 -6662.475,E2 -6662.475} C_VEL
LIN {X 0,Y 488.207,Z 382.517,A -85,B 0,C 180,E1 -6663.3,E2 -6663.3} C_VEL
LIN {X 0,Y 488.386,Z 379.208,A -85,B 0,C 180,E1 -6664.125,E2 -6664.125} C_VEL
LIN {X 0,Y 488.483,Z 373.777,A -85,B 0,C 180,E1 -6665.158,E2 -6665.158} C_VEL
LIN {X 0,Y 488.543,Z 367.965,A -85,B 0,C 180,E1 -6665.985,E2 -6665.985} C_VEL
LIN {X 0,Y 488.689,Z 360.758,A -85,B 0,C 180,E1 -6666.795,E2 -6666.795} C_VEL
LIN {X 0,Y 488.816,Z 353.323,A -85,B 0,C 180,E1 -6667.434,E2 -6667.434} C_VEL
LIN {X 0,Y 489.017,Z 343.815,A -85,B 0,C 180,E1 -6668.054,E2 -6668.054} C_VEL
LIN {X 0,Y 488.811,Z 335.962,A -85,B 0,C 180,E1 -6668.421,E2 -6668.421} C_VEL
LIN {X 0,Y 488.239,Z 332.246,A -85,B 0,C 180,E1 -6668.588,E2 -6668.588} C_VEL
LIN {X 0,Y 488.315,Z 324.58,A -85,B 0,C 180,E1 -6671.851,E2 -6671.851} C_VEL
LIN {X 0,Y 488.347,Z 316.366,A -85,B 0,C 180,E1 -6675.371,E2 -6675.371} C_VEL
LIN {X 0,Y 488.413,Z 308.195,A -85,B 0,C 180,E1 -6678.889,E2 -6678.889} C_VEL
LIN {X 0,Y 488.423,Z 302.027,A -85,B 0,C 180,E1 -6681.525,E2 -6681.525} C_VEL
LIN {X 0,Y 488.476,Z 294.716,A -85,B 0,C 180,E1 -6684.659,E2 -6684.659} C_VEL
LIN {X 0,Y 488.558,Z 287.056,A -85,B 0,C 180,E1 -6687.872,E2 -6687.872} C_VEL
LIN {X 0,Y 488.653,Z 283.62,A -85,B 0,C 180,E1 -6689.332,E2 -6689.332} C_VEL
LIN {X 0,Y 488.684,Z 283.608,A -85,B 0,C 180,E1 -6692.147,E2 -6692.147} C_VEL
LIN {X 0,Y 488.706,Z 283.613,A -85,B 0,C 180,E1 -6695.114,E2 -6695.114} C_VEL
LIN {X 0,Y 488.668,Z 283.611,A -85,B 0,C 180,E1 -6698.199,E2 -6698.199} C_VEL
LIN {X 0,Y 488.673,Z 283.612,A -85,B 0,C 180,E1 -6701.417,E2 -6701.417} C_VEL
LIN {X 0,Y 488.693,Z 283.614,A -85,B 0,C 180,E1 -6704.802,E2 -6704.802} C_VEL
LIN {X 0,Y 488.683,Z 283.61,A -85,B 0,C 180,E1 -6707.473,E2 -6707.473} C_VEL
LIN {X 0,Y 488.724,Z 283.606,A -85,B 0,C 180,E1 -6709.675,E2 -6709.675} C_VEL
LIN {X 0,Y 488.674,Z 283.612,A -85,B 0,C 180,E1 -6712.84,E2 -6712.84} C_VEL
LIN {X 0,Y 488.726,Z 283.609,A -85,B 0,C 180,E1 -6715.887,E2 -6715.887} C_VEL
LIN {X 0,Y 488.687,Z 283.61,A -85,B 0,C 180,E1 -6718.82,E2 -6718.82} C_VEL
LIN {X 0,Y 488.737,Z 283.607,A -85,B 0,C 180,E1 -6721.671,E2 -6721.671} C_VEL
LIN {X 0,Y 488.757,Z 283.605,A -85,B 0,C 180,E1 -6723.504,E2 -6723.504} C_VEL
LIN {X 0,Y 488.077,Z 283.692,A -85,B 0,C 180,E1 -6724.192,E2 -6724.192} C_VEL
LIN {X 0,Y 485.209,Z 284.05,A -85,B 0,C 180,E1 -6725.308,E2 -6725.308} C_VEL
LIN {X 0,Y 482.782,Z 284.349,A -85,B 0,C 180,E1 -6726.209,E2 -6726.209} C_VEL
LIN {X 0,Y 481.731,Z 284.48,A -85,B 0,C 180,E1 -6726.904,E2 -6726.904} C_VEL
LIN {X 0,Y 481.641,Z 284.488,A -85,B 0,C 180,E1 -6727.14,E2 -6727.14} C_VEL
LIN {X 0,Y 481.686,Z 284.485,A -85,B 0,C 180,E1 -6729.502,E2 -6729.502} C_VEL
LIN {X 0,Y 481.695,Z 284.481,A -85,B 0,C 180,E1 -6732.158,E2 -6732.158} C_VEL
LIN {X 0,Y 481.73,Z 284.481,A -85,B 0,C 180,E1 -6734.775,E2 -6734.775} C_VEL
LIN {X 0,Y 481.738,Z 284.478,A -85,B 0,C 180,E1 -6738.215,E2 -6738.215} C_VEL
LIN {X 0,Y 481.727,Z 284.476,A -85,B 0,C 180,E1 -6741.611,E2 -6741.611} C_VEL
LIN {X 0,Y 481.781,Z 284.474,A -85,B 0,C 180,E1 -6744.139,E2 -6744.139} C_VEL
LIN {X 0,Y 481.896,Z 284.455,A -85,B 0,C 180,E1 -6747.492,E2 -6747.492} C_VEL
LIN {X 0,Y 481.897,Z 284.462,A -85,B 0,C 180,E1 -6750,E2 -6750} C_VEL
LIN {X 0,Y 481.897,Z 284.455,A -85,B 0,C 180,E1 -6752.508,E2 -6752.508} C_VEL
LIN {X 0,Y 481.781,Z 284.474,A -85,B 0,C 180,E1 -6755.861,E2 -6755.861} C_VEL
LIN {X 0,Y 481.727,Z 284.476,A -85,B 0,C 180,E1 -6758.389,E2 -6758.389} C_VEL
LIN {X 0,Y 481.738,Z 284.477,A -85,B 0,C 180,E1 -6761.785,E2 -6761.785} C_VEL
LIN {X 0,Y 481.73,Z 284.481,A -85,B 0,C 180,E1 -6765.225,E2 -6765.225} C_VEL
LIN {X 0,Y 481.701,Z 284.483,A -85,B 0,C 180,E1 -6768.722,E2 -6768.722} C_VEL
LIN {X 0,Y 481.636,Z 284.49,A -85,B 0,C 180,E1 -6771.395,E2 -6771.395} C_VEL
LIN {X 0,Y 481.667,Z 284.487,A -85,B 0,C 180,E1 -6774.114,E2 -6774.114} C_VEL
LIN {X 0,Y 481.742,Z 284.476,A -85,B 0,C 180,E1 -6777.141,E2 -6777.141} C_VEL
LIN {X 0,Y 481.678,Z 284.485,A -85,B 0,C 180,E1 -6779.741,E2 -6779.741} C_VEL
LIN {X 0,Y 481.664,Z 284.487,A -85,B 0,C 180,E1 -6782.675,E2 -6782.675} C_VEL
LIN {X 0,Y 481.634,Z 284.494,A -85,B 0,C 180,E1 -6785.71,E2 -6785.71} C_VEL
LIN {X 0,Y 481.663,Z 284.485,A -85,B 0,C 180,E1 -6788.86,E2 -6788.86} C_VEL
LIN {X 0,Y 481.645,Z 284.489,A -85,B 0,C 180,E1 -6791.914,E2 -6791.914} C_VEL
LIN {X 0,Y 481.647,Z 284.486,A -85,B 0,C 180,E1 -6794.459,E2 -6794.459} C_VEL
LIN {X 0,Y 481.632,Z 284.489,A -85,B 0,C 180,E1 -6797.84,E2 -6797.84} C_VEL
LIN {X 0,Y 481.659,Z 284.489,A -85,B 0,C 180,E1 -6801.142,E2 -6801.142} C_VEL
LIN {X 0,Y 481.649,Z 284.492,A -85,B 0,C 180,E1 -6804.798,E2 -6804.798} C_VEL
LIN {X 0,Y 481.643,Z 284.485,A -85,B 0,C 180,E1 -6807.814,E2 -6807.814} C_VEL
LIN {X 0,Y 481.767,Z 284.64,A -85,B 0,C 180,E1 -6809.784,E2 -6809.784} C_VEL
LIN {X 0,Y 481.672,Z 289.54,A -85,B 0,C 180,E1 -6812.168,E2 -6812.168} C_VEL
LIN {X 0,Y 481.504,Z 295.294,A -85,B 0,C 180,E1 -6814.96,E2 -6814.96} C_VEL
LIN {X 0,Y 481.381,Z 301.05,A -85,B 0,C 180,E1 -6817.693,E2 -6817.693} C_VEL
LIN {X 0,Y 481.308,Z 306.733,A -85,B 0,C 180,E1 -6820.378,E2 -6820.378} C_VEL
LIN {X 0,Y 481.191,Z 312.393,A -85,B 0,C 180,E1 -6823.017,E2 -6823.017} C_VEL
LIN {X 0,Y 481.105,Z 318.04,A -85,B 0,C 180,E1 -6825.622,E2 -6825.622} C_VEL
LIN {X 0,Y 481.113,Z 323.675,A -85,B 0,C 180,E1 -6828.2,E2 -6828.2} C_VEL
LIN {X 0,Y 481.019,Z 330.09,A -85,B 0,C 180,E1 -6831.097,E2 -6831.097} C_VEL
LIN {X 0,Y 482.26,Z 340.083,A -85,B 0,C 180,E1 -6831.569,E2 -6831.569} C_VEL
LIN {X 0,Y 482.012,Z 349.63,A -85,B 0,C 180,E1 -6832.145,E2 -6832.145} C_VEL
LIN {X 0,Y 481.818,Z 358.19,A -85,B 0,C 180,E1 -6832.838,E2 -6832.838} C_VEL
LIN {X 0,Y 481.568,Z 366.476,A -85,B 0,C 180,E1 -6833.717,E2 -6833.717} C_VEL
LIN {X 0,Y 481.545,Z 372.59,A -85,B 0,C 180,E1 -6834.558,E2 -6834.558} C_VEL
LIN {X 0,Y 481.375,Z 378.499,A -85,B 0,C 180,E1 -6835.605,E2 -6835.605} C_VEL
LIN {X 0,Y 481.162,Z 382.869,A -85,B 0,C 180,E1 -6836.652,E2 -6836.652} C_VEL
LIN {X 0,Y 481.01,Z 385.449,A -85,B 0,C 180,E1 -6837.489,E2 -6837.489} C_VEL
LIN {X 0,Y 480.937,Z 387.276,A -85,B 0,C 180,E1 -6838.326,E2 -6838.326} C_VEL
LIN {X 0,Y 480.925,Z 388.402,A -85,B 0,C 180,E1 -6839.164,E2 -6839.164} C_VEL
LIN {X 0,Y 480.928,Z 388.857,A -85,B 0,C 180,E1 -6840.001,E2 -6840.001} C_VEL
LIN {X 0,Y 480.938,Z 388.647,A -85,B 0,C 180,E1 -6840.838,E2 -6840.838} C_VEL
LIN {X 0,Y 480.967,Z 387.769,A -85,B 0,C 180,E1 -6841.676,E2 -6841.676} C_VEL
LIN {X 0,Y 481.227,Z 385.13,A -85,B 0,C 180,E1 -6842.931,E2 -6842.931} C_VEL
LIN {X 0,Y 481.401,Z 382.43,A -85,B 0,C 180,E1 -6843.768,E2 -6843.768} C_VEL
LIN {X 0,Y 481.456,Z 377.899,A -85,B 0,C 180,E1 -6844.816,E2 -6844.816} C_VEL
LIN {X 0,Y 481.623,Z 371.755,A -85,B 0,C 180,E1 -6845.864,E2 -6845.864} C_VEL
LIN {X 0,Y 481.81,Z 364.217,A -85,B 0,C 180,E1 -6846.836,E2 -6846.836} C_VEL
LIN {X 0,Y 482.169,Z 356.211,A -85,B 0,C 180,E1 -6847.624,E2 -6847.624} C_VEL
LIN {X 0,Y 482.334,Z 347.858,A -85,B 0,C 180,E1 -6848.263,E2 -6848.263} C_VEL
LIN {X 0,Y 482.402,Z 338.548,A -85,B 0,C 180,E1 -6848.8,E2 -6848.8} C_VEL
LIN {X 0,Y 481.193,Z 331.69,A -85,B 0,C 180,E1 -6849.14,E2 -6849.14} C_VEL
LIN {X 0,Y 481.296,Z 325.722,A -85,B 0,C 180,E1 -6851.943,E2 -6851.943} C_VEL
LIN {X 0,Y 481.462,Z 318.202,A -85,B 0,C 180,E1 -6855.545,E2 -6855.545} C_VEL
LIN {X 0,Y 481.606,Z 311.732,A -85,B 0,C 180,E1 -6858.727,E2 -6858.727} C_VEL
LIN {X 0,Y 481.776,Z 306.377,A -85,B 0,C 180,E1 -6861.39,E2 -6861.39} C_VEL
LIN {X 0,Y 481.913,Z 300.922,A -85,B 0,C 180,E1 -6864.101,E2 -6864.101} C_VEL
LIN {X 0,Y 482.143,Z 295.554,A -85,B 0,C 180,E1 -6866.865,E2 -6866.865} C_VEL
LIN {X 0,Y 482.321,Z 290.225,A -85,B 0,C 180,E1 -6869.698,E2 -6869.698} C_VEL
LIN {X 0,Y 482.041,Z 286.714,A -85,B 0,C 180,E1 -6871.66,E2 -6871.66} C_VEL
LIN {X 0,Y 481.708,Z 284.485,A -85,B 0,C 180,E1 -6873.045,E2 -6873.045} C_VEL
LIN {X 0,Y 481.642,Z 284.493,A -85,B 0,C 180,E1 -6875.71,E2 -6875.71} C_VEL
LIN {X 0,Y 481.676,Z 284.488,A -85,B 0,C 180,E1 -6878.86,E2 -6878.86} C_VEL
LIN {X 0,Y 481.658,Z 284.491,A -85,B 0,C 180,E1 -6881.913,E2 -6881.913} C_VEL
LIN {X 0,Y 481.66,Z 284.491,A -85,B 0,C 180,E1 -6884.458,E2 -6884.458} C_VEL
LIN {X 0,Y 481.653,Z 284.491,A -85,B 0,C 180,E1 -6887.84,E2 -6887.84} C_VEL
LIN {X 0,Y 481.685,Z 284.488,A -85,B 0,C 180,E1 -6890.652,E2 -6890.652} C_VEL
LIN {X 0,Y 481.632,Z 284.494,A -85,B 0,C 180,E1 -6893.376,E2 -6893.376} C_VEL
LIN {X 0,Y 481.711,Z 284.672,A -85,B 0,C 180,E1 -6895.7,E2 -6895.7} C_VEL
LIN {X 0,Y 482.917,Z 289.707,A -85,B 0,C 180,E1 -6897.575,E2 -6897.575} C_VEL
LIN {X 0,Y 484.611,Z 297.308,A -85,B 0,C 180,E1 -6899.978,E2 -6899.978} C_VEL
LIN {X 0,Y 485.275,Z 300.826,A -85,B 0,C 180,E1 -6900.977,E2 -6900.977} C_VEL
LIN {X 0,Y 485.116,Z 305.271,A -85,B 0,C 180,E1 -6902.096,E2 -6902.096} C_VEL
LIN {X 0,Y 483.975,Z 317.294,A -85,B 0,C 180,E1 -6904.865,E2 -6904.865} C_VEL
LIN {X 0,Y 482.989,Z 332.975,A -85,B 0,C 180,E1 -6908.22,E2 -6908.22} C_VEL
LIN {X 0,Y 482.259,Z 348.833,A -85,B 0,C 180,E1 -6911.415,E2 -6911.415} C_VEL
LIN {X 0,Y 481.789,Z 364.522,A -85,B 0,C 180,E1 -6914.442,E2 -6914.442} C_VEL
LIN {X 0,Y 481.705,Z 369.393,A -85,B 0,C 180,E1 -6915.369,E2 -6915.369} C_VEL
LIN {X 0,Y 483.061,Z 383.219,A -85,B 0,C 180,E1 -6915.721,E2 -6915.721} C_VEL
LIN {X 0,Y 483.238,Z 389.387,A -85,B 0,C 180,E1 -6915.927,E2 -6915.927} C_VEL
LIN {X 0,Y 482.922,Z 402.365,A -85,B 0,C 180,E1 -6916.481,E2 -6916.481} C_VEL
LIN {X 0,Y 482.533,Z 414.177,A -85,B 0,C 180,E1 -6917.167,E2 -6917.167} C_VEL
LIN {X 0,Y 482.235,Z 426.083,A -85,B 0,C 180,E1 -6918.052,E2 -6918.052} C_VEL
LIN {X 0,Y 481.865,Z 435.857,A -85,B 0,C 180,E1 -6918.964,E2 -6918.964} C_VEL
LIN {X 0,Y 481.456,Z 445.919,A -85,B 0,C 180,E1 -6920.124,E2 -6920.124} C_VEL
LIN {X 0,Y 481.279,Z 453.397,A -85,B 0,C 180,E1 -6921.18,E2 -6921.18} C_VEL
LIN {X 0,Y 481.117,Z 460.727,A -85,B 0,C 180,E1 -6922.445,E2 -6922.445} C_VEL
LIN {X 0,Y 480.969,Z 466.842,A -85,B 0,C 180,E1 -6923.785,E2 -6923.785} C_VEL
LIN {X 0,Y 480.914,Z 471.102,A -85,B 0,C 180,E1 -6924.97,E2 -6924.97} C_VEL
LIN {X 0,Y 481.002,Z 473.522,A -85,B 0,C 180,E1 -6925.81,E2 -6925.81} C_VEL
LIN {X 0,Y 480.996,Z 475.487,A -85,B 0,C 180,E1 -6926.649,E2 -6926.649} C_VEL
LIN {X 0,Y 480.941,Z 476.964,A -85,B 0,C 180,E1 -6927.487,E2 -6927.487} C_VEL
LIN {X 0,Y 480.828,Z 478.658,A -85,B 0,C 180,E1 -6929.163,E2 -6929.163} C_VEL
LIN {X 0,Y 480.83,Z 478.902,A -85,B 0,C 180,E1 -6930,E2 -6930} C_VEL
LIN {X 0,Y 480.825,Z 478.692,A -85,B 0,C 180,E1 -6930.837,E2 -6930.837} C_VEL
LIN {X 0,Y 480.94,Z 477.081,A -85,B 0,C 180,E1 -6932.513,E2 -6932.513} C_VEL
LIN {X 0,Y 480.981,Z 475.633,A -85,B 0,C 180,E1 -6933.351,E2 -6933.351} C_VEL
LIN {X 0,Y 480.895,Z 472.604,A -85,B 0,C 180,E1 -6934.61,E2 -6934.61} C_VEL
LIN {X 0,Y 481.012,Z 468.499,A -85,B 0,C 180,E1 -6935.87,E2 -6935.87} C_VEL
LIN {X 0,Y 481.108,Z 462.154,A -85,B 0,C 180,E1 -6937.344,E2 -6937.344} C_VEL
LIN {X 0,Y 481.282,Z 455.224,A -85,B 0,C 180,E1 -6938.608,E2 -6938.608} C_VEL
LIN {X 0,Y 481.418,Z 448.116,A -85,B 0,C 180,E1 -6939.665,E2 -6939.665} C_VEL
LIN {X 0,Y 481.725,Z 439.516,A -85,B 0,C 180,E1 -6940.72,E2 -6940.72} C_VEL
LIN {X 0,Y 482.134,Z 428.867,A -85,B 0,C 180,E1 -6941.775,E2 -6941.775} C_VEL
LIN {X 0,Y 482.45,Z 418.277,A -85,B 0,C 180,E1 -6942.622,E2 -6942.622} C_VEL
LIN {X 0,Y 482.843,Z 406.516,A -85,B 0,C 180,E1 -6943.36,E2 -6943.36} C_VEL
LIN {X 0,Y 483.201,Z 394.281,A -85,B 0,C 180,E1 -6943.939,E2 -6943.939} C_VEL
LIN {X 0,Y 483.239,Z 384.01,A -85,B 0,C 180,E1 -6944.301,E2 -6944.301} C_VEL
LIN {X 0,Y 481.826,Z 370.666,A -85,B 0,C 180,E1 -6944.644,E2 -6944.644} C_VEL
LIN {X 0,Y 481.756,Z 369.806,A -85,B 0,C 180,E1 -6944.683,E2 -6944.683} C_VEL
LIN {X 0,Y 482.278,Z 352.492,A -85,B 0,C 180,E1 -6948.039,E2 -6948.039} C_VEL
LIN {X 0,Y 482.959,Z 335.695,A -85,B 0,C 180,E1 -6951.356,E2 -6951.356} C_VEL
LIN {X 0,Y 483.871,Z 318.107,A -85,B 0,C 180,E1 -6954.911,E2 -6954.911} C_VEL
LIN {X 0,Y 484.935,Z 301.598,A -85,B 0,C 180,E1 -6958.351,E2 -6958.351} C_VEL
LIN {X 0,Y 484.706,Z 298.38,A -85,B 0,C 180,E1 -6959.061,E2 -6959.061} C_VEL
LIN {X 0,Y 482.024,Z 286.256,A -85,B 0,C 180,E1 -6961.924,E2 -6961.924} C_VEL
LIN {X 0,Y 481.669,Z 284.488,A -85,B 0,C 180,E1 -6962.393,E2 -6962.393} C_VEL
LIN {X 0,Y 481.665,Z 284.49,A -85,B 0,C 180,E1 -6965.204,E2 -6965.204} C_VEL
LIN {X 0,Y 481.66,Z 284.49,A -85,B 0,C 180,E1 -6968.007,E2 -6968.007} C_VEL
LIN {X 0,Y 481.661,Z 284.488,A -85,B 0,C 180,E1 -6971.042,E2 -6971.042} C_VEL
LIN {X 0,Y 481.665,Z 284.488,A -85,B 0,C 180,E1 -6974.457,E2 -6974.457} C_VEL
LIN {X 0,Y 481.653,Z 284.491,A -85,B 0,C 180,E1 -6977.839,E2 -6977.839} C_VEL
LIN {X 0,Y 481.686,Z 284.486,A -85,B 0,C 180,E1 -6980.651,E2 -6980.651} C_VEL
LIN {X 0,Y 481.633,Z 284.494,A -85,B 0,C 180,E1 -6983.376,E2 -6983.376} C_VEL
LIN {X 0,Y 481.682,Z 284.489,A -85,B 0,C 180,E1 -6986.327,E2 -6986.327} C_VEL
LIN {X 0,Y 481.628,Z 284.496,A -85,B 0,C 180,E1 -6989.423,E2 -6989.423} C_VEL
LIN {X 0,Y 481.474,Z 284.602,A -85,B 0,C 180,E1 -6991.679,E2 -6991.679} C_VEL
LIN {X 0,Y 481.455,Z 293.366,A -85,B 0,C 180,E1 -6994.829,E2 -6994.829} C_VEL
LIN {X 0,Y 481.431,Z 300.911,A -85,B 0,C 180,E1 -6997.693,E2 -6997.693} C_VEL
LIN {X 0,Y 481.442,Z 307.68,A -85,B 0,C 180,E1 -7000.381,E2 -7000.381} C_VEL
LIN {X 0,Y 481.375,Z 315.099,A -85,B 0,C 180,E1 -7003.458,E2 -7003.458} C_VEL
LIN {X 0,Y 481.338,Z 321.431,A -85,B 0,C 180,E1 -7006.058,E2 -7006.058} C_VEL
LIN {X 0,Y 481.361,Z 327.494,A -85,B 0,C 180,E1 -7008.631,E2 -7008.631} C_VEL
LIN {X 0,Y 481.354,Z 334.08,A -85,B 0,C 180,E1 -7011.392,E2 -7011.392} C_VEL
LIN {X 0,Y 482.112,Z 340.468,A -85,B 0,C 180,E1 -7011.67,E2 -7011.67} C_VEL
LIN {X 0,Y 481.978,Z 349.005,A -85,B 0,C 180,E1 -7012.142,E2 -7012.142} C_VEL
LIN {X 0,Y 481.87,Z 356.904,A -85,B 0,C 180,E1 -7012.717,E2 -7012.717} C_VEL
LIN {X 0,Y 481.541,Z 365.003,A -85,B 0,C 180,E1 -7013.504,E2 -7013.504} C_VEL
LIN {X 0,Y 481.609,Z 371.66,A -85,B 0,C 180,E1 -7014.346,E2 -7014.346} C_VEL
